KUKA KRL program: EPS_2_25716_MHCF01_A_20250828082512.src

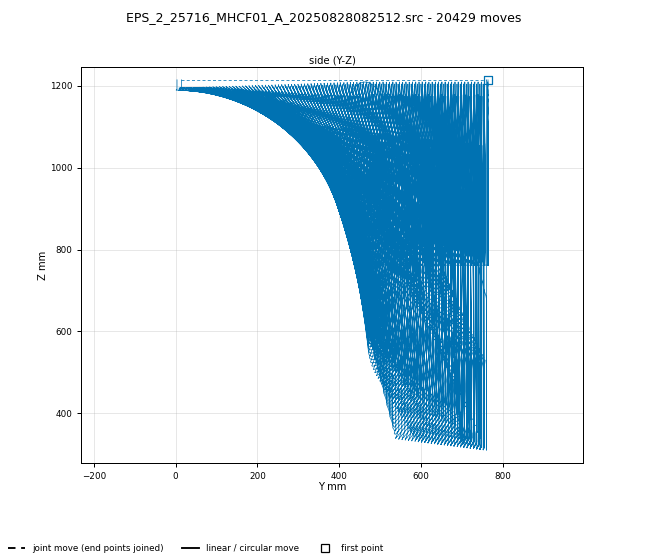
[picture p0: tool path of EPS_2_25716_MHCF01_A_20250828082512.src, 20429 of 20431 moves have a stored position in this frame; points joined in program order, loops and branches not executed]
&ACCESS RVP
&REL 4
&COMMENT QRS 19112012
&PARAM EDITMASK = *
DEF PART()
EXT BAS (BAS_COMMAND :IN,REAL :IN )
INT I
BAS (#INITMOV,0 )

;KUKA QRS Post kuka4.cps  Date:22-06-2017 !

File_ID=2800

QRS_PRE_INIT()

;Init var - Until changes are made in qrs_pre_init
Outlet_Square_prg=0
Inlet_1_Square_prg=0
Inlet_2_Square_prg=0
Inlet_3_Square_prg=0
Inlet_4_Square_prg=0
Inlet_5_Square_prg=0

Outlet_1={X 0.000, Y 457.000, Z 786.000, B 0.000, E1 0.000 }
Inlet_1={X 0.000, Y 688.000, Z 484.500, B 0.000, E1 109.000 }
Inlet_2={X 0.000, Y 457.000, Z 756.000, B 0.000, E1 180.000 }
Outlet_1_type=838
Inlet_1_type=201
Inlet_2_type=838
;QRS#1=Sidecore dimensions
;QRS#2=825-33" Concrete
;QRS#3=200-8" PVC SDR 35
;QRS#4=825-33" Concrete
;QRS#5=
;QRS#6=
;QRS#7=
;QRS#8=
;QRS#9=S306-46
;QRS#10=12-08 PSX
;QRS#11=S306-46
;QRS#12=
;QRS#13=
;QRS#14=
;QRS#15=
;QRS#16=1524x152x1676 5,5'
;QRS#17=EPS Height
;QRS#18=1205
;QRS#19=*
;QRS#20= UPDATED VERSION 22-06-2017
;QRS#21=*
Outlet_Square=0650
Inlet_1_Square=0100
Inlet_2_Square=0650
Inlet_3_Square=0
Inlet_4_Square=0
Inlet_5_Square=0
Mill_Square=1
Outlet_Square_Prg=267
Inlet_1_Square_prg=204
Inlet_2_Square_prg=267

QRS_INIT()

$ADVANCE=5

; T1
PTP {E1 176.359,E2 176.359}
PTP {X 0,Y 763.722,A -85,B 0,C 180,E1 176.359,E2 176.359,E3 0,E4 0,E5 0,E6 0}
QRS_SPEED_INIT()
LIN {X 0,Y 763.722,Z 1215,A -85,B 0,C 180,E1 176.359,E2 176.359,E3 0,E4 0,E5 0,E6 0} C_VEL
LIN {X 0,Y 763.722,Z 764.06,A -85,B 0,C 180,E1 176.359,E2 176.359} C_VEL
LIN {X 0,Y 763.74,Z 762.06,A -85,B 0,C 180,E1 176.509,E2 176.509} C_VEL
LIN {X 0,Y 763.887,Z 762.06,A -85,B 0,C 180,E1 177.187,E2 177.187} C_VEL
LIN {X 0,Y 763.859,Z 762.06,A -85,B 0,C 180,E1 184.692,E2 184.692} C_VEL
LIN {X 0,Y 763.829,Z 762.06,A -85,B 0,C 180,E1 192.28,E2 192.28} C_VEL
LIN {X 0,Y 763.844,Z 762.06,A -85,B 0,C 180,E1 200.095,E2 200.095} C_VEL
LIN {X 0,Y 763.817,Z 762.06,A -85,B 0,C 180,E1 208.325,E2 208.325} C_VEL
LIN {X 0,Y 762.405,Z 762.06,A -85,B 0,C 180,E1 210.54,E2 210.54} C_VEL
LIN {X 0,Y 762.716,Z 762.06,A -85,B 0,C 180,E1 214.993,E2 214.993} C_VEL
LIN {X 0,Y 763.716,Z 762.06,A -85,B 0,C 180,E1 216.696,E2 216.696} C_VEL
LIN {X 0,Y 763.502,Z 762.06,A -85,B 0,C 180,E1 224.735,E2 224.735} C_VEL
LIN {X 0,Y 763.769,Z 762.06,A -85,B 0,C 180,E1 225.284,E2 225.284} C_VEL
LIN {X 0,Y 763.693,Z 762.06,A -85,B 0,C 180,E1 233.306,E2 233.306} C_VEL
LIN {X 0,Y 763.603,Z 762.06,A -85,B 0,C 180,E1 233.585,E2 233.585} C_VEL
LIN {X 0,Y 763.11,Z 765.125,A -85,B 0,C 180,E1 233.691,E2 233.691} C_VEL
LIN {X 0,Y 763.161,Z 825.383,A -85,B 0,C 180,E1 234.39,E2 234.39} C_VEL
LIN {X 0,Y 763.585,Z 842.967,A -85,B 0,C 180,E1 234.683,E2 234.683} C_VEL
LIN {X 0,Y 763.687,Z 860.331,A -85,B 0,C 180,E1 235.017,E2 235.017} C_VEL
LIN {X 0,Y 763.614,Z 876.794,A -85,B 0,C 180,E1 235.382,E2 235.382} C_VEL
LIN {X 0,Y 763.265,Z 892.83,A -85,B 0,C 180,E1 235.785,E2 235.785} C_VEL
LIN {X 0,Y 763.632,Z 912.821,A -85,B 0,C 180,E1 236.407,E2 236.407} C_VEL
LIN {X 0,Y 763.653,Z 925.004,A -85,B 0,C 180,E1 236.825,E2 236.825} C_VEL
LIN {X 0,Y 763.67,Z 937.193,A -85,B 0,C 180,E1 237.266,E2 237.266} C_VEL
LIN {X 0,Y 763.647,Z 955.469,A -85,B 0,C 180,E1 238,E2 238} C_VEL
LIN {X 0,Y 763.481,Z 968.04,A -85,B 0,C 180,E1 238.551,E2 238.551} C_VEL
LIN {X 0,Y 763.562,Z 976.639,A -85,B 0,C 180,E1 238.958,E2 238.958} C_VEL
LIN {X 0,Y 763.516,Z 991.054,A -85,B 0,C 180,E1 239.67,E2 239.67} C_VEL
LIN {X 0,Y 763.481,Z 1008.327,A -85,B 0,C 180,E1 240.607,E2 240.607} C_VEL
LIN {X 0,Y 763.638,Z 1024.574,A -85,B 0,C 180,E1 241.577,E2 241.577} C_VEL
LIN {X 0,Y 763.597,Z 1040.363,A -85,B 0,C 180,E1 242.593,E2 242.593} C_VEL
LIN {X 0,Y 763.3,Z 1055.407,A -85,B 0,C 180,E1 243.633,E2 243.633} C_VEL
LIN {X 0,Y 763.19,Z 1070.044,A -85,B 0,C 180,E1 244.738,E2 244.738} C_VEL
LIN {X 0,Y 763.448,Z 1083.451,A -85,B 0,C 180,E1 245.843,E2 245.843} C_VEL
LIN {X 0,Y 763.685,Z 1096.507,A -85,B 0,C 180,E1 247.002,E2 247.002} C_VEL
LIN {X 0,Y 763.164,Z 1110.017,A -85,B 0,C 180,E1 248.281,E2 248.281} C_VEL
LIN {X 0,Y 762.922,Z 1121.794,A -85,B 0,C 180,E1 249.496,E2 249.496} C_VEL
LIN {X 0,Y 763.257,Z 1133.579,A -85,B 0,C 180,E1 250.838,E2 250.838} C_VEL
LIN {X 0,Y 763.827,Z 1143.997,A -85,B 0,C 180,E1 252.134,E2 252.134} C_VEL
LIN {X 0,Y 763.056,Z 1154.828,A -85,B 0,C 180,E1 253.589,E2 253.589} C_VEL
LIN {X 0,Y 762.742,Z 1164.591,A -85,B 0,C 180,E1 255.058,E2 255.058} C_VEL
LIN {X 0,Y 763.115,Z 1172.356,A -85,B 0,C 180,E1 256.36,E2 256.36} C_VEL
LIN {X 0,Y 763.85,Z 1179.543,A -85,B 0,C 180,E1 257.719,E2 257.719} C_VEL
LIN {X 0,Y 762.886,Z 1187.41,A -85,B 0,C 180,E1 259.379,E2 259.379} C_VEL
LIN {X 0,Y 762.625,Z 1192.228,A -85,B 0,C 180,E1 260.568,E2 260.568} C_VEL
LIN {X 0,Y 762.79,Z 1195.671,A -85,B 0,C 180,E1 261.52,E2 261.52} C_VEL
LIN {X 0,Y 763.28,Z 1198.709,A -85,B 0,C 180,E1 262.473,E2 262.473} C_VEL
LIN {X 0,Y 763.858,Z 1201.341,A -85,B 0,C 180,E1 263.423,E2 263.423} C_VEL
LIN {X 0,Y 763.267,Z 1203.655,A -85,B 0,C 180,E1 264.361,E2 264.361} C_VEL
LIN {X 0,Y 762.79,Z 1205.61,A -85,B 0,C 180,E1 265.3,E2 265.3} C_VEL
LIN {X 0,Y 762.61,Z 1207.2,A -85,B 0,C 180,E1 266.241,E2 266.241} C_VEL
LIN {X 0,Y 762.976,Z 1208.861,A -85,B 0,C 180,E1 267.626,E2 267.626} C_VEL
LIN {X 0,Y 763.872,Z 1209.666,A -85,B 0,C 180,E1 269.062,E2 269.062} C_VEL
LIN {X 0,Y 762.824,Z 1209.715,A -85,B 0,C 180,E1 270.938,E2 270.938} C_VEL
LIN {X 0,Y 762.626,Z 1209.464,A -85,B 0,C 180,E1 271.62,E2 271.62} C_VEL
LIN {X 0,Y 762.799,Z 1208.403,A -85,B 0,C 180,E1 272.816,E2 272.816} C_VEL
LIN {X 0,Y 763.271,Z 1207.186,A -85,B 0,C 180,E1 273.754,E2 273.754} C_VEL
LIN {X 0,Y 763.867,Z 1205.578,A -85,B 0,C 180,E1 274.691,E2 274.691} C_VEL
LIN {X 0,Y 763.013,Z 1202.59,A -85,B 0,C 180,E1 276.11,E2 276.11} C_VEL
LIN {X 0,Y 762.637,Z 1198.719,A -85,B 0,C 180,E1 277.532,E2 277.532} C_VEL
LIN {X 0,Y 762.799,Z 1195.679,A -85,B 0,C 180,E1 278.478,E2 278.478} C_VEL
LIN {X 0,Y 763.569,Z 1190.402,A -85,B 0,C 180,E1 279.894,E2 279.894} C_VEL
LIN {X 0,Y 763.864,Z 1188.414,A -85,B 0,C 180,E1 280.366,E2 280.366} C_VEL
LIN {X 0,Y 763.206,Z 1182.988,A -85,B 0,C 180,E1 281.57,E2 281.57} C_VEL
LIN {X 0,Y 762.859,Z 1179.555,A -85,B 0,C 180,E1 282.295,E2 282.295} C_VEL
LIN {X 0,Y 762.736,Z 1172.088,A -85,B 0,C 180,E1 283.694,E2 283.694} C_VEL
LIN {X 0,Y 763.29,Z 1163.914,A -85,B 0,C 180,E1 285.044,E2 285.044} C_VEL
LIN {X 0,Y 763.763,Z 1158.345,A -85,B 0,C 180,E1 285.87,E2 285.87} C_VEL
LIN {X 0,Y 763.637,Z 1154.843,A -85,B 0,C 180,E1 286.396,E2 286.396} C_VEL
LIN {X 0,Y 762.912,Z 1144.015,A -85,B 0,C 180,E1 287.885,E2 287.885} C_VEL
LIN {X 0,Y 762.868,Z 1131.999,A -85,B 0,C 180,E1 289.358,E2 289.358} C_VEL
LIN {X 0,Y 763.42,Z 1120.427,A -85,B 0,C 180,E1 290.638,E2 290.638} C_VEL
LIN {X 0,Y 763.768,Z 1112.188,A -85,B 0,C 180,E1 291.477,E2 291.477} C_VEL
LIN {X 0,Y 763.558,Z 1105.867,A -85,B 0,C 180,E1 292.112,E2 292.112} C_VEL
LIN {X 0,Y 763.217,Z 1095.124,A -85,B 0,C 180,E1 293.139,E2 293.139} C_VEL
LIN {X 0,Y 763.157,Z 1081.838,A -85,B 0,C 180,E1 294.303,E2 294.303} C_VEL
LIN {X 0,Y 763.464,Z 1068.233,A -85,B 0,C 180,E1 295.394,E2 295.394} C_VEL
LIN {X 0,Y 763.661,Z 1053.626,A -85,B 0,C 180,E1 296.482,E2 296.482} C_VEL
LIN {X 0,Y 763.464,Z 1037.389,A -85,B 0,C 180,E1 297.608,E2 297.608} C_VEL
LIN {X 0,Y 763.397,Z 1021.761,A -85,B 0,C 180,E1 298.604,E2 298.604} C_VEL
LIN {X 0,Y 763.561,Z 1005.354,A -85,B 0,C 180,E1 299.557,E2 299.557} C_VEL
LIN {X 0,Y 763.593,Z 989.474,A -85,B 0,C 180,E1 300.41,E2 300.41} C_VEL
LIN {X 0,Y 763.623,Z 970.492,A -85,B 0,C 180,E1 301.334,E2 301.334} C_VEL
LIN {X 0,Y 763.591,Z 951.717,A -85,B 0,C 180,E1 302.16,E2 302.16} C_VEL
LIN {X 0,Y 763.583,Z 933.277,A -85,B 0,C 180,E1 302.887,E2 302.887} C_VEL
LIN {X 0,Y 763.349,Z 920.518,A -85,B 0,C 180,E1 303.348,E2 303.348} C_VEL
LIN {X 0,Y 763.571,Z 911.94,A -85,B 0,C 180,E1 303.623,E2 303.623} C_VEL
LIN {X 0,Y 763.721,Z 893.155,A -85,B 0,C 180,E1 304.183,E2 304.183} C_VEL
LIN {X 0,Y 763.708,Z 877.523,A -85,B 0,C 180,E1 304.595,E2 304.595} C_VEL
LIN {X 0,Y 763.535,Z 860.886,A -85,B 0,C 180,E1 304.979,E2 304.979} C_VEL
LIN {X 0,Y 763.204,Z 848.058,A -85,B 0,C 180,E1 305.249,E2 305.249} C_VEL
LIN {X 0,Y 763.489,Z 831.034,A -85,B 0,C 180,E1 305.511,E2 305.511} C_VEL
LIN {X 0,Y 763.515,Z 819.053,A -85,B 0,C 180,E1 305.669,E2 305.669} C_VEL
LIN {X 0,Y 763.118,Z 762.451,A -85,B 0,C 180,E1 306.339,E2 306.339} C_VEL
LIN {X 0,Y 763.741,Z 762.06,A -85,B 0,C 180,E1 306.442,E2 306.442} C_VEL
LIN {X 0,Y 763.705,Z 762.06,A -85,B 0,C 180,E1 306.695,E2 306.695} C_VEL
LIN {X 0,Y 763.761,Z 762.06,A -85,B 0,C 180,E1 314.713,E2 314.713} C_VEL
LIN {X 0,Y 763.525,Z 762.06,A -85,B 0,C 180,E1 315.267,E2 315.267} C_VEL
LIN {X 0,Y 762.411,Z 762.06,A -85,B 0,C 180,E1 320.387,E2 320.387} C_VEL
LIN {X 0,Y 763.765,Z 762.06,A -85,B 0,C 180,E1 322.742,E2 322.742} C_VEL
LIN {X 0,Y 763.828,Z 762.06,A -85,B 0,C 180,E1 329.523,E2 329.523} C_VEL
LIN {X 0,Y 763.838,Z 762.06,A -85,B 0,C 180,E1 335.857,E2 335.857} C_VEL
LIN {X 0,Y 763.844,Z 762.06,A -85,B 0,C 180,E1 343.851,E2 343.851} C_VEL
LIN {X 0,Y 763.841,Z 762.06,A -85,B 0,C 180,E1 351.533,E2 351.533} C_VEL
LIN {X 0,Y 763.874,Z 762.06,A -85,B 0,C 180,E1 359.063,E2 359.063} C_VEL
LIN {X 0,Y 763.873,Z 762.06,A -85,B 0,C 180,E1 366.576,E2 366.576} C_VEL
LIN {X 0,Y 763.842,Z 762.06,A -85,B 0,C 180,E1 374.206,E2 374.206} C_VEL
LIN {X 0,Y 763.813,Z 762.06,A -85,B 0,C 180,E1 382.105,E2 382.105} C_VEL
LIN {X 0,Y 762.966,Z 762.06,A -85,B 0,C 180,E1 388.36,E2 388.36} C_VEL
LIN {X 0,Y 763.69,Z 762.06,A -85,B 0,C 180,E1 389.858,E2 389.858} C_VEL
LIN {X 0,Y 763.788,Z 762.06,A -85,B 0,C 180,E1 397.257,E2 397.257} C_VEL
LIN {X 0,Y 762.288,Z 762.06,A -85,B 0,C 180,E1 402.464,E2 402.464} C_VEL
LIN {X 0,Y 763.518,Z 762.06,A -85,B 0,C 180,E1 404.734,E2 404.734} C_VEL
LIN {X 0,Y 763.738,Z 762.06,A -85,B 0,C 180,E1 405.285,E2 405.285} C_VEL
LIN {X 0,Y 763.711,Z 762.06,A -85,B 0,C 180,E1 413.304,E2 413.304} C_VEL
LIN {X 0,Y 763.665,Z 762.06,A -85,B 0,C 180,E1 413.601,E2 413.601} C_VEL
LIN {X 0,Y 761.693,Z 762.06,A -85,B 0,C 180,E1 413.812,E2 413.812} C_VEL
LIN {X 0,Y 761.807,Z 763.834,A -85,B 0,C 180,E1 413.903,E2 413.903} C_VEL
LIN {X 0,Y 762.762,Z 766.677,A -85,B 0,C 180,E1 413.987,E2 413.987} C_VEL
LIN {X 0,Y 763.131,Z 768.605,A -85,B 0,C 180,E1 414.029,E2 414.029} C_VEL
LIN {X 0,Y 763.648,Z 798.138,A -85,B 0,C 180,E1 414.411,E2 414.411} C_VEL
LIN {X 0,Y 763.664,Z 815.21,A -85,B 0,C 180,E1 414.679,E2 414.679} C_VEL
LIN {X 0,Y 763.409,Z 832.281,A -85,B 0,C 180,E1 414.998,E2 414.998} C_VEL
LIN {X 0,Y 763.24,Z 839.694,A -85,B 0,C 180,E1 415.153,E2 415.153} C_VEL
LIN {X 0,Y 763.609,Z 855.772,A -85,B 0,C 180,E1 415.565,E2 415.565} C_VEL
LIN {X 0,Y 763.663,Z 868.895,A -85,B 0,C 180,E1 415.935,E2 415.935} C_VEL
LIN {X 0,Y 763.644,Z 887.88,A -85,B 0,C 180,E1 416.529,E2 416.529} C_VEL
LIN {X 0,Y 763.368,Z 905.889,A -85,B 0,C 180,E1 417.155,E2 417.155} C_VEL
LIN {X 0,Y 763.602,Z 925.254,A -85,B 0,C 180,E1 417.944,E2 417.944} C_VEL
LIN {X 0,Y 763.603,Z 943.443,A -85,B 0,C 180,E1 418.758,E2 418.758} C_VEL
LIN {X 0,Y 763.642,Z 961.593,A -85,B 0,C 180,E1 419.66,E2 419.66} C_VEL
LIN {X 0,Y 763.586,Z 977.603,A -85,B 0,C 180,E1 420.524,E2 420.524} C_VEL
LIN {X 0,Y 763.415,Z 994.185,A -85,B 0,C 180,E1 421.498,E2 421.498} C_VEL
LIN {X 0,Y 763.335,Z 1011.042,A -85,B 0,C 180,E1 422.585,E2 422.585} C_VEL
LIN {X 0,Y 763.547,Z 1026.034,A -85,B 0,C 180,E1 423.645,E2 423.645} C_VEL
LIN {X 0,Y 763.647,Z 1040.062,A -85,B 0,C 180,E1 424.711,E2 424.711} C_VEL
LIN {X 0,Y 763.256,Z 1053.988,A -85,B 0,C 180,E1 425.839,E2 425.839} C_VEL
LIN {X 0,Y 763.018,Z 1067.004,A -85,B 0,C 180,E1 426.983,E2 426.983} C_VEL
LIN {X 0,Y 763.297,Z 1080.095,A -85,B 0,C 180,E1 428.248,E2 428.248} C_VEL
LIN {X 0,Y 763.803,Z 1092.173,A -85,B 0,C 180,E1 429.518,E2 429.518} C_VEL
LIN {X 0,Y 763.199,Z 1103.736,A -85,B 0,C 180,E1 430.811,E2 430.811} C_VEL
LIN {X 0,Y 762.791,Z 1114.347,A -85,B 0,C 180,E1 432.112,E2 432.112} C_VEL
LIN {X 0,Y 763.102,Z 1125.142,A -85,B 0,C 180,E1 433.592,E2 433.592} C_VEL
LIN {X 0,Y 763.761,Z 1133.68,A -85,B 0,C 180,E1 434.882,E2 434.882} C_VEL
LIN {X 0,Y 763.673,Z 1136.311,A -85,B 0,C 180,E1 435.318,E2 435.318} C_VEL
LIN {X 0,Y 762.988,Z 1143.295,A -85,B 0,C 180,E1 436.488,E2 436.488} C_VEL
LIN {X 0,Y 762.6,Z 1150.963,A -85,B 0,C 180,E1 437.941,E2 437.941} C_VEL
LIN {X 0,Y 763.021,Z 1157.607,A -85,B 0,C 180,E1 439.383,E2 439.383} C_VEL
LIN {X 0,Y 763.734,Z 1162.407,A -85,B 0,C 180,E1 440.584,E2 440.584} C_VEL
LIN {X 0,Y 763.71,Z 1164.155,A -85,B 0,C 180,E1 441.058,E2 441.058} C_VEL
LIN {X 0,Y 763.145,Z 1167.372,A -85,B 0,C 180,E1 442,E2 442} C_VEL
LIN {X 0,Y 762.743,Z 1170.222,A -85,B 0,C 180,E1 442.943,E2 442.943} C_VEL
LIN {X 0,Y 762.645,Z 1172.699,A -85,B 0,C 180,E1 443.887,E2 443.887} C_VEL
LIN {X 0,Y 763.158,Z 1175.695,A -85,B 0,C 180,E1 445.305,E2 445.305} C_VEL
LIN {X 0,Y 763.838,Z 1177.41,A -85,B 0,C 180,E1 446.389,E2 446.389} C_VEL
LIN {X 0,Y 763.399,Z 1178.43,A -85,B 0,C 180,E1 447.186,E2 447.186} C_VEL
LIN {X 0,Y 762.558,Z 1179.735,A -85,B 0,C 180,E1 449.062,E2 449.062} C_VEL
LIN {X 0,Y 762.983,Z 1179.696,A -85,B 0,C 180,E1 450.94,E2 450.94} C_VEL
LIN {X 0,Y 763.578,Z 1178.326,A -85,B 0,C 180,E1 452.815,E2 452.815} C_VEL
LIN {X 0,Y 763.007,Z 1177.129,A -85,B 0,C 180,E1 453.757,E2 453.757} C_VEL
LIN {X 0,Y 762.687,Z 1175.523,A -85,B 0,C 180,E1 454.7,E2 454.7} C_VEL
LIN {X 0,Y 762.806,Z 1172.471,A -85,B 0,C 180,E1 456.114,E2 456.114} C_VEL
LIN {X 0,Y 763.563,Z 1168.572,A -85,B 0,C 180,E1 457.525,E2 457.525} C_VEL
LIN {X 0,Y 763.871,Z 1167.062,A -85,B 0,C 180,E1 457.994,E2 457.994} C_VEL
LIN {X 0,Y 763.298,Z 1163.834,A -85,B 0,C 180,E1 458.949,E2 458.949} C_VEL
LIN {X 0,Y 762.809,Z 1160.211,A -85,B 0,C 180,E1 459.906,E2 459.906} C_VEL
LIN {X 0,Y 762.632,Z 1156.118,A -85,B 0,C 180,E1 460.863,E2 460.863} C_VEL
LIN {X 0,Y 763.012,Z 1149.302,A -85,B 0,C 180,E1 462.295,E2 462.295} C_VEL
LIN {X 0,Y 763.742,Z 1142.426,A -85,B 0,C 180,E1 463.571,E2 463.571} C_VEL
LIN {X 0,Y 763.77,Z 1140.524,A -85,B 0,C 180,E1 463.889,E2 463.889} C_VEL
LIN {X 0,Y 763.149,Z 1133.842,A -85,B 0,C 180,E1 465.014,E2 465.014} C_VEL
LIN {X 0,Y 762.72,Z 1124.527,A -85,B 0,C 180,E1 466.419,E2 466.419} C_VEL
LIN {X 0,Y 763.111,Z 1112.649,A -85,B 0,C 180,E1 468.006,E2 468.006} C_VEL
LIN {X 0,Y 763.786,Z 1101.998,A -85,B 0,C 180,E1 469.289,E2 469.289} C_VEL
LIN {X 0,Y 763.295,Z 1090.039,A -85,B 0,C 180,E1 470.636,E2 470.636} C_VEL
LIN {X 0,Y 762.981,Z 1078.156,A -85,B 0,C 180,E1 471.867,E2 471.867} C_VEL
LIN {X 0,Y 763.239,Z 1064.584,A -85,B 0,C 180,E1 473.14,E2 473.14} C_VEL
LIN {X 0,Y 763.68,Z 1051.16,A -85,B 0,C 180,E1 474.295,E2 474.295} C_VEL
LIN {X 0,Y 763.565,Z 1039.109,A -85,B 0,C 180,E1 475.278,E2 475.278} C_VEL
LIN {X 0,Y 763.278,Z 1022.943,A -85,B 0,C 180,E1 476.498,E2 476.498} C_VEL
LIN {X 0,Y 763.364,Z 1007.682,A -85,B 0,C 180,E1 477.548,E2 477.548} C_VEL
LIN {X 0,Y 763.578,Z 991.976,A -85,B 0,C 180,E1 478.539,E2 478.539} C_VEL
LIN {X 0,Y 763.634,Z 974.917,A -85,B 0,C 180,E1 479.532,E2 479.532} C_VEL
LIN {X 0,Y 763.542,Z 958.559,A -85,B 0,C 180,E1 480.413,E2 480.413} C_VEL
LIN {X 0,Y 763.571,Z 940.113,A -85,B 0,C 180,E1 481.309,E2 481.309} C_VEL
LIN {X 0,Y 763.536,Z 921.233,A -85,B 0,C 180,E1 482.137,E2 482.137} C_VEL
LIN {X 0,Y 763.431,Z 914.252,A -85,B 0,C 180,E1 482.419,E2 482.419} C_VEL
LIN {X 0,Y 763.666,Z 902.086,A -85,B 0,C 180,E1 482.879,E2 482.879} C_VEL
LIN {X 0,Y 763.698,Z 884.096,A -85,B 0,C 180,E1 483.505,E2 483.505} C_VEL
LIN {X 0,Y 763.64,Z 863.566,A -85,B 0,C 180,E1 484.131,E2 484.131} C_VEL
LIN {X 0,Y 763.324,Z 846.79,A -85,B 0,C 180,E1 484.588,E2 484.588} C_VEL
LIN {X 0,Y 763.327,Z 841.786,A -85,B 0,C 180,E1 484.704,E2 484.704} C_VEL
LIN {X 0,Y 763.694,Z 825.562,A -85,B 0,C 180,E1 485.036,E2 485.036} C_VEL
LIN {X 0,Y 763.758,Z 807.93,A -85,B 0,C 180,E1 485.347,E2 485.347} C_VEL
LIN {X 0,Y 763.695,Z 792.713,A -85,B 0,C 180,E1 485.569,E2 485.569} C_VEL
LIN {X 0,Y 763.223,Z 767.95,A -85,B 0,C 180,E1 485.883,E2 485.883} C_VEL
LIN {X 0,Y 763.265,Z 762.06,A -85,B 0,C 180,E1 485.98,E2 485.98} C_VEL
LIN {X 0,Y 763.595,Z 762.06,A -85,B 0,C 180,E1 486.6,E2 486.6} C_VEL
LIN {X 0,Y 763.808,Z 762.06,A -85,B 0,C 180,E1 492.131,E2 492.131} C_VEL
LIN {X 0,Y 763.614,Z 762.06,A -85,B 0,C 180,E1 492.57,E2 492.57} C_VEL
LIN {X 0,Y 763.875,Z 762.06,A -85,B 0,C 180,E1 500.258,E2 500.258} C_VEL
LIN {X 0,Y 763.733,Z 762.06,A -85,B 0,C 180,E1 506.566,E2 506.566} C_VEL
LIN {X 0,Y 763.499,Z 762.06,A -85,B 0,C 180,E1 507.306,E2 507.306} C_VEL
LIN {X 0,Y 763.209,Z 762.122,A -85,B 0,C 180,E1 507.486,E2 507.486} C_VEL
LIN {X 0,Y 763.638,Z 763.12,A -85,B 0,C 180,E1 507.53,E2 507.53} C_VEL
LIN {X 0,Y 763.79,Z 765.738,A -85,B 0,C 180,E1 507.626,E2 507.626} C_VEL
LIN {X 0,Y 763.797,Z 831.68,A -85,B 0,C 180,E1 509.978,E2 509.978} C_VEL
LIN {X 0,Y 763.29,Z 835.99,A -85,B 0,C 180,E1 510.124,E2 510.124} C_VEL
LIN {X 0,Y 763.012,Z 837.649,A -85,B 0,C 180,E1 510.172,E2 510.172} C_VEL
LIN {X 0,Y 763.701,Z 916.034,A -85,B 0,C 180,E1 510.916,E2 510.916} C_VEL
LIN {X 0,Y 763.838,Z 948.168,A -85,B 0,C 180,E1 511.225,E2 511.225} C_VEL
LIN {X 0,Y 763.826,Z 957.76,A -85,B 0,C 180,E1 511.354,E2 511.354} C_VEL
LIN {X 0,Y 763.852,Z 968.842,A -85,B 0,C 180,E1 511.58,E2 511.58} C_VEL
LIN {X 0,Y 763.85,Z 979.495,A -85,B 0,C 180,E1 511.875,E2 511.875} C_VEL
LIN {X 0,Y 763.751,Z 990.547,A -85,B 0,C 180,E1 512.269,E2 512.269} C_VEL
LIN {X 0,Y 763.666,Z 1000.84,A -85,B 0,C 180,E1 512.728,E2 512.728} C_VEL
LIN {X 0,Y 763.853,Z 1010.575,A -85,B 0,C 180,E1 513.262,E2 513.262} C_VEL
LIN {X 0,Y 763.738,Z 1018.552,A -85,B 0,C 180,E1 513.781,E2 513.781} C_VEL
LIN {X 0,Y 763.337,Z 1026.8,A -85,B 0,C 180,E1 514.414,E2 514.414} C_VEL
LIN {X 0,Y 763.391,Z 1034.378,A -85,B 0,C 180,E1 515.117,E2 515.117} C_VEL
LIN {X 0,Y 763.816,Z 1040.943,A -85,B 0,C 180,E1 515.856,E2 515.856} C_VEL
LIN {X 0,Y 763.73,Z 1044.687,A -85,B 0,C 180,E1 516.366,E2 516.366} C_VEL
LIN {X 0,Y 763.556,Z 1046.498,A -85,B 0,C 180,E1 516.616,E2 516.616} C_VEL
LIN {X 0,Y 763.126,Z 1051.588,A -85,B 0,C 180,E1 517.493,E2 517.493} C_VEL
LIN {X 0,Y 763.403,Z 1055.387,A -85,B 0,C 180,E1 518.38,E2 518.38} C_VEL
LIN {X 0,Y 763.87,Z 1057.915,A -85,B 0,C 180,E1 519.233,E2 519.233} C_VEL
LIN {X 0,Y 763.413,Z 1059.478,A -85,B 0,C 180,E1 520.109,E2 520.109} C_VEL
LIN {X 0,Y 763.251,Z 1059.957,A -85,B 0,C 180,E1 521.032,E2 521.032} C_VEL
LIN {X 0,Y 763.655,Z 1059.354,A -85,B 0,C 180,E1 521.885,E2 521.885} C_VEL
LIN {X 0,Y 763.862,Z 1058.461,A -85,B 0,C 180,E1 522.382,E2 522.382} C_VEL
LIN {X 0,Y 763.738,Z 1058.034,A -85,B 0,C 180,E1 522.625,E2 522.625} C_VEL
LIN {X 0,Y 763.24,Z 1055.162,A -85,B 0,C 180,E1 523.594,E2 523.594} C_VEL
LIN {X 0,Y 763.303,Z 1051.925,A -85,B 0,C 180,E1 524.344,E2 524.344} C_VEL
LIN {X 0,Y 763.727,Z 1047.737,A -85,B 0,C 180,E1 525.09,E2 525.09} C_VEL
LIN {X 0,Y 763.841,Z 1046.258,A -85,B 0,C 180,E1 525.326,E2 525.326} C_VEL
LIN {X 0,Y 763.734,Z 1040.569,A -85,B 0,C 180,E1 526.099,E2 526.099} C_VEL
LIN {X 0,Y 763.771,Z 1035.105,A -85,B 0,C 180,E1 526.714,E2 526.714} C_VEL
LIN {X 0,Y 763.809,Z 1027.112,A -85,B 0,C 180,E1 527.466,E2 527.466} C_VEL
LIN {X 0,Y 763.493,Z 1019.373,A -85,B 0,C 180,E1 528.074,E2 528.074} C_VEL
LIN {X 0,Y 763.527,Z 1010.215,A -85,B 0,C 180,E1 528.673,E2 528.673} C_VEL
LIN {X 0,Y 763.845,Z 1000.103,A -85,B 0,C 180,E1 529.215,E2 529.215} C_VEL
LIN {X 0,Y 763.796,Z 989.571,A -85,B 0,C 180,E1 529.678,E2 529.678} C_VEL
LIN {X 0,Y 763.682,Z 979.025,A -85,B 0,C 180,E1 530.051,E2 530.051} C_VEL
LIN {X 0,Y 763.841,Z 967.337,A -85,B 0,C 180,E1 530.364,E2 530.364} C_VEL
LIN {X 0,Y 763.864,Z 955.826,A -85,B 0,C 180,E1 530.586,E2 530.586} C_VEL
LIN {X 0,Y 763.864,Z 944.689,A -85,B 0,C 180,E1 530.724,E2 530.724} C_VEL
LIN {X 0,Y 763.795,Z 840.857,A -85,B 0,C 180,E1 531.697,E2 531.697} C_VEL
LIN {X 0,Y 763.395,Z 837.234,A -85,B 0,C 180,E1 531.74,E2 531.74} C_VEL
LIN {X 0,Y 763.377,Z 762.06,A -85,B 0,C 180,E1 534.427,E2 534.427} C_VEL
LIN {X 0,Y 763.879,Z 762.06,A -85,B 0,C 180,E1 534.598,E2 534.598} C_VEL
LIN {X 0,Y 763.74,Z 762.06,A -85,B 0,C 180,E1 536.509,E2 536.509} C_VEL
LIN {X 0,Y 754.649,Z 762.06,A -85,B 0,C 180,E1 539.103,E2 539.103} C_VEL
LIN {X 0,Y 754.714,Z 762.06,A -85,B 0,C 180,E1 546.382,E2 546.382} C_VEL
LIN {X 0,Y 754.951,Z 762.06,A -85,B 0,C 180,E1 553.398,E2 553.398} C_VEL
LIN {X 0,Y 755.106,Z 762.06,A -85,B 0,C 180,E1 560.956,E2 560.956} C_VEL
LIN {X 0,Y 754.907,Z 762.06,A -85,B 0,C 180,E1 569.538,E2 569.538} C_VEL
LIN {X 0,Y 754.747,Z 762.06,A -85,B 0,C 180,E1 577.859,E2 577.859} C_VEL
LIN {X 0,Y 755.038,Z 762.06,A -85,B 0,C 180,E1 586.149,E2 586.149} C_VEL
LIN {X 0,Y 755.772,Z 763.476,A -85,B 0,C 180,E1 593.262,E2 593.262} C_VEL
LIN {X 0,Y 757.071,Z 866.865,A -85,B 0,C 180,E1 594.806,E2 594.806} C_VEL
LIN {X 0,Y 756.764,Z 937.982,A -85,B 0,C 180,E1 596.961,E2 596.961} C_VEL
LIN {X 0,Y 756.208,Z 1009.087,A -85,B 0,C 180,E1 600.342,E2 600.342} C_VEL
LIN {X 0,Y 755.591,Z 1073.769,A -85,B 0,C 180,E1 604.774,E2 604.774} C_VEL
LIN {X 0,Y 755.159,Z 1125.985,A -85,B 0,C 180,E1 609.753,E2 609.753} C_VEL
LIN {X 0,Y 754.885,Z 1162.64,A -85,B 0,C 180,E1 614.586,E2 614.586} C_VEL
LIN {X 0,Y 754.929,Z 1187.619,A -85,B 0,C 180,E1 619.317,E2 619.317} C_VEL
LIN {X 0,Y 755.011,Z 1204.817,A -85,B 0,C 180,E1 624.842,E2 624.842} C_VEL
LIN {X 0,Y 755.6,Z 1209.848,A -85,B 0,C 180,E1 629.455,E2 629.455} C_VEL
LIN {X 0,Y 755.213,Z 1203.673,A -85,B 0,C 180,E1 635.696,E2 635.696} C_VEL
LIN {X 0,Y 755.209,Z 1183.325,A -85,B 0,C 180,E1 641.622,E2 641.622} C_VEL
LIN {X 0,Y 755.279,Z 1149.721,A -85,B 0,C 180,E1 647.293,E2 647.293} C_VEL
LIN {X 0,Y 755.616,Z 1101.536,A -85,B 0,C 180,E1 652.773,E2 652.773} C_VEL
LIN {X 0,Y 756.053,Z 1041.761,A -85,B 0,C 180,E1 657.605,E2 657.605} C_VEL
LIN {X 0,Y 756.539,Z 972.654,A -85,B 0,C 180,E1 661.561,E2 661.561} C_VEL
LIN {X 0,Y 756.981,Z 899.217,A -85,B 0,C 180,E1 664.352,E2 664.352} C_VEL
LIN {X 0,Y 757.033,Z 825.171,A -85,B 0,C 180,E1 665.945,E2 665.945} C_VEL
LIN {X 0,Y 755.604,Z 762.06,A -85,B 0,C 180,E1 666.801,E2 666.801} C_VEL
LIN {X 0,Y 754.964,Z 762.06,A -85,B 0,C 180,E1 676.058,E2 676.058} C_VEL
LIN {X 0,Y 755.187,Z 762.06,A -85,B 0,C 180,E1 683.61,E2 683.61} C_VEL
LIN {X 0,Y 754.991,Z 762.06,A -85,B 0,C 180,E1 691.018,E2 691.018} C_VEL
LIN {X 0,Y 754.99,Z 762.06,A -85,B 0,C 180,E1 696.892,E2 696.892} C_VEL
LIN {X 0,Y 755.509,Z 762.06,A -85,B 0,C 180,E1 704.234,E2 704.234} C_VEL
LIN {X 0,Y 755.149,Z 762.06,A -85,B 0,C 180,E1 712.462,E2 712.462} C_VEL
LIN {X 0,Y 754.843,Z 762.06,A -85,B 0,C 180,E1 720.542,E2 720.542} C_VEL
LIN {X 0,Y 755.16,Z 762.06,A -85,B 0,C 180,E1 727.47,E2 727.47} C_VEL
LIN {X 0,Y 754.722,Z 762.06,A -85,B 0,C 180,E1 735.712,E2 735.712} C_VEL
LIN {X 0,Y 755.109,Z 762.06,A -85,B 0,C 180,E1 743.031,E2 743.031} C_VEL
LIN {X 0,Y 754.738,Z 762.06,A -85,B 0,C 180,E1 751.245,E2 751.245} C_VEL
LIN {X 0,Y 755.372,Z 762.06,A -85,B 0,C 180,E1 757.737,E2 757.737} C_VEL
LIN {X 0,Y 755.086,Z 762.06,A -85,B 0,C 180,E1 766.068,E2 766.068} C_VEL
LIN {X 0,Y 754.847,Z 762.617,A -85,B 0,C 180,E1 773.503,E2 773.503} C_VEL
LIN {X 0,Y 756.838,Z 851.222,A -85,B 0,C 180,E1 775.096,E2 775.096} C_VEL
LIN {X 0,Y 756.572,Z 927.019,A -85,B 0,C 180,E1 777.689,E2 777.689} C_VEL
LIN {X 0,Y 756.03,Z 997.6,A -85,B 0,C 180,E1 781.416,E2 781.416} C_VEL
LIN {X 0,Y 755.498,Z 1059.465,A -85,B 0,C 180,E1 786.063,E2 786.063} C_VEL
LIN {X 0,Y 755.207,Z 1107.459,A -85,B 0,C 180,E1 791.064,E2 791.064} C_VEL
LIN {X 0,Y 755.121,Z 1143.123,A -85,B 0,C 180,E1 796.312,E2 796.312} C_VEL
LIN {X 0,Y 755.209,Z 1167.271,A -85,B 0,C 180,E1 801.884,E2 801.884} C_VEL
LIN {X 0,Y 755.441,Z 1178.391,A -85,B 0,C 180,E1 807.091,E2 807.091} C_VEL
LIN {X 0,Y 755.577,Z 1178.361,A -85,B 0,C 180,E1 812.847,E2 812.847} C_VEL
LIN {X 0,Y 755.337,Z 1164.251,A -85,B 0,C 180,E1 818.926,E2 818.926} C_VEL
LIN {X 0,Y 755.313,Z 1136.006,A -85,B 0,C 180,E1 824.809,E2 824.809} C_VEL
LIN {X 0,Y 755.571,Z 1094.24,A -85,B 0,C 180,E1 830.389,E2 830.389} C_VEL
LIN {X 0,Y 755.949,Z 1039.354,A -85,B 0,C 180,E1 835.532,E2 835.532} C_VEL
LIN {X 0,Y 756.379,Z 973.926,A -85,B 0,C 180,E1 839.899,E2 839.899} C_VEL
LIN {X 0,Y 756.794,Z 902.312,A -85,B 0,C 180,E1 843.209,E2 843.209} C_VEL
LIN {X 0,Y 757.059,Z 828.537,A -85,B 0,C 180,E1 845.328,E2 845.328} C_VEL
LIN {X 0,Y 755.501,Z 762.06,A -85,B 0,C 180,E1 846.417,E2 846.417} C_VEL
LIN {X 0,Y 754.691,Z 762.06,A -85,B 0,C 180,E1 853.876,E2 853.876} C_VEL
LIN {X 0,Y 755.508,Z 762.06,A -85,B 0,C 180,E1 860.801,E2 860.801} C_VEL
LIN {X 0,Y 755.399,Z 762.845,A -85,B 0,C 180,E1 867.37,E2 867.37} C_VEL
LIN {X 0,Y 755.203,Z 841.66,A -85,B 0,C 180,E1 870.097,E2 870.097} C_VEL
LIN {X 0,Y 755.975,Z 969.088,A -85,B 0,C 180,E1 871.489,E2 871.489} C_VEL
LIN {X 0,Y 755.852,Z 1007.886,A -85,B 0,C 180,E1 873.027,E2 873.027} C_VEL
LIN {X 0,Y 755.636,Z 1038.476,A -85,B 0,C 180,E1 875.515,E2 875.515} C_VEL
LIN {X 0,Y 755.532,Z 1056.178,A -85,B 0,C 180,E1 878.603,E2 878.603} C_VEL
LIN {X 0,Y 755.659,Z 1059.384,A -85,B 0,C 180,E1 881.903,E2 881.903} C_VEL
LIN {X 0,Y 755.786,Z 1047.355,A -85,B 0,C 180,E1 885.205,E2 885.205} C_VEL
LIN {X 0,Y 755.593,Z 1021.178,A -85,B 0,C 180,E1 888.01,E2 888.01} C_VEL
LIN {X 0,Y 755.835,Z 985.532,A -85,B 0,C 180,E1 889.918,E2 889.918} C_VEL
LIN {X 0,Y 755.981,Z 944.278,A -85,B 0,C 180,E1 890.831,E2 890.831} C_VEL
LIN {X 0,Y 755.464,Z 831.48,A -85,B 0,C 180,E1 892.061,E2 892.061} C_VEL
LIN {X 0,Y 755.867,Z 762.06,A -85,B 0,C 180,E1 894.707,E2 894.707} C_VEL
LIN {X 0,Y 754.649,Z 762.06,A -85,B 0,C 180,E1 899.103,E2 899.103} C_VEL
LIN {X 0,Y 746.34,Z 762.06,A -85,B 0,C 180,E1 901.736,E2 901.736} C_VEL
LIN {X 0,Y 746.674,Z 762.06,A -85,B 0,C 180,E1 906.451,E2 906.451} C_VEL
LIN {X 0,Y 746.854,Z 762.06,A -85,B 0,C 180,E1 913.546,E2 913.546} C_VEL
LIN {X 0,Y 747.186,Z 762.06,A -85,B 0,C 180,E1 920.852,E2 920.852} C_VEL
LIN {X 0,Y 747.493,Z 762.06,A -85,B 0,C 180,E1 928.528,E2 928.528} C_VEL
LIN {X 0,Y 747.254,Z 762.06,A -85,B 0,C 180,E1 936.839,E2 936.839} C_VEL
LIN {X 0,Y 746.997,Z 762.06,A -85,B 0,C 180,E1 946.191,E2 946.191} C_VEL
LIN {X 0,Y 747.444,Z 763.808,A -85,B 0,C 180,E1 952.788,E2 952.788} C_VEL
LIN {X 0,Y 750.231,Z 776.864,A -85,B 0,C 180,E1 953.103,E2 953.103} C_VEL
LIN {X 0,Y 750.506,Z 865.678,A -85,B 0,C 180,E1 954.425,E2 954.425} C_VEL
LIN {X 0,Y 749.923,Z 935.971,A -85,B 0,C 180,E1 956.538,E2 956.538} C_VEL
LIN {X 0,Y 748.996,Z 1006.584,A -85,B 0,C 180,E1 959.878,E2 959.878} C_VEL
LIN {X 0,Y 748.022,Z 1071.537,A -85,B 0,C 180,E1 964.313,E2 964.313} C_VEL
LIN {X 0,Y 747.303,Z 1123.291,A -85,B 0,C 180,E1 969.22,E2 969.22} C_VEL
LIN {X 0,Y 747.011,Z 1160.66,A -85,B 0,C 180,E1 974.117,E2 974.117} C_VEL
LIN {X 0,Y 746.988,Z 1187.62,A -85,B 0,C 180,E1 979.202,E2 979.202} C_VEL
LIN {X 0,Y 747.047,Z 1204.817,A -85,B 0,C 180,E1 984.787,E2 984.787} C_VEL
LIN {X 0,Y 747.593,Z 1209.85,A -85,B 0,C 180,E1 989.449,E2 989.449} C_VEL
LIN {X 0,Y 747.473,Z 1204.698,A -85,B 0,C 180,E1 995.272,E2 995.272} C_VEL
LIN {X 0,Y 747.343,Z 1184.684,A -85,B 0,C 180,E1 1001.449,E2 1001.449} C_VEL
LIN {X 0,Y 747.377,Z 1150.917,A -85,B 0,C 180,E1 1007.317,E2 1007.317} C_VEL
LIN {X 0,Y 747.89,Z 1102.898,A -85,B 0,C 180,E1 1012.889,E2 1012.889} C_VEL
LIN {X 0,Y 748.614,Z 1043.481,A -85,B 0,C 180,E1 1017.781,E2 1017.781} C_VEL
LIN {X 0,Y 749.445,Z 974.583,A -85,B 0,C 180,E1 1021.798,E2 1021.798} C_VEL
LIN {X 0,Y 750.189,Z 902.678,A -85,B 0,C 180,E1 1024.598,E2 1024.598} C_VEL
LIN {X 0,Y 750.501,Z 828.692,A -85,B 0,C 180,E1 1026.256,E2 1026.256} C_VEL
LIN {X 0,Y 748.648,Z 766.444,A -85,B 0,C 180,E1 1027.111,E2 1027.111} C_VEL
LIN {X 0,Y 747.086,Z 762.06,A -85,B 0,C 180,E1 1027.435,E2 1027.435} C_VEL
LIN {X 0,Y 746.891,Z 762.06,A -85,B 0,C 180,E1 1036.198,E2 1036.198} C_VEL
LIN {X 0,Y 746.758,Z 762.06,A -85,B 0,C 180,E1 1044.574,E2 1044.574} C_VEL
LIN {X 0,Y 746.854,Z 762.06,A -85,B 0,C 180,E1 1051.445,E2 1051.445} C_VEL
LIN {X 0,Y 746.526,Z 762.06,A -85,B 0,C 180,E1 1057.72,E2 1057.72} C_VEL
LIN {X 0,Y 746.822,Z 762.06,A -85,B 0,C 180,E1 1065.253,E2 1065.253} C_VEL
LIN {X 0,Y 747.172,Z 762.06,A -85,B 0,C 180,E1 1072.381,E2 1072.381} C_VEL
LIN {X 0,Y 746.857,Z 762.06,A -85,B 0,C 180,E1 1080.548,E2 1080.548} C_VEL
LIN {X 0,Y 747.097,Z 762.06,A -85,B 0,C 180,E1 1087.551,E2 1087.551} C_VEL
LIN {X 0,Y 747.089,Z 762.06,A -85,B 0,C 180,E1 1095.146,E2 1095.146} C_VEL
LIN {X 0,Y 746.946,Z 762.06,A -85,B 0,C 180,E1 1103.297,E2 1103.297} C_VEL
LIN {X 0,Y 746.794,Z 762.06,A -85,B 0,C 180,E1 1111.164,E2 1111.164} C_VEL
LIN {X 0,Y 746.849,Z 762.06,A -85,B 0,C 180,E1 1118.489,E2 1118.489} C_VEL
LIN {X 0,Y 747.06,Z 762.06,A -85,B 0,C 180,E1 1126.087,E2 1126.087} C_VEL
LIN {X 0,Y 747.766,Z 763.987,A -85,B 0,C 180,E1 1133.117,E2 1133.117} C_VEL
LIN {X 0,Y 750.587,Z 792.853,A -85,B 0,C 180,E1 1133.623,E2 1133.623} C_VEL
LIN {X 0,Y 750.25,Z 865.72,A -85,B 0,C 180,E1 1135.143,E2 1135.143} C_VEL
LIN {X 0,Y 749.515,Z 936.849,A -85,B 0,C 180,E1 1137.796,E2 1137.796} C_VEL
LIN {X 0,Y 748.585,Z 1005.86,A -85,B 0,C 180,E1 1141.649,E2 1141.649} C_VEL
LIN {X 0,Y 747.69,Z 1066.56,A -85,B 0,C 180,E1 1146.441,E2 1146.441} C_VEL
LIN {X 0,Y 747.167,Z 1112.549,A -85,B 0,C 180,E1 1151.492,E2 1151.492} C_VEL
LIN {X 0,Y 747.055,Z 1144.678,A -85,B 0,C 180,E1 1156.461,E2 1156.461} C_VEL
LIN {X 0,Y 747.273,Z 1167.268,A -85,B 0,C 180,E1 1161.797,E2 1161.797} C_VEL
LIN {X 0,Y 747.441,Z 1178.391,A -85,B 0,C 180,E1 1167.06,E2 1167.06} C_VEL
LIN {X 0,Y 747.546,Z 1178.362,A -85,B 0,C 180,E1 1172.878,E2 1172.878} C_VEL
LIN {X 0,Y 747.284,Z 1164.254,A -85,B 0,C 180,E1 1179.022,E2 1179.022} C_VEL
LIN {X 0,Y 747.355,Z 1136.677,A -85,B 0,C 180,E1 1184.857,E2 1184.857} C_VEL
LIN {X 0,Y 747.764,Z 1095.593,A -85,B 0,C 180,E1 1190.456,E2 1190.456} C_VEL
LIN {X 0,Y 748.338,Z 1040.471,A -85,B 0,C 180,E1 1195.72,E2 1195.72} C_VEL
LIN {X 0,Y 749.131,Z 975.529,A -85,B 0,C 180,E1 1200.13,E2 1200.13} C_VEL
LIN {X 0,Y 749.918,Z 903.828,A -85,B 0,C 180,E1 1203.498,E2 1203.498} C_VEL
LIN {X 0,Y 750.478,Z 829.13,A -85,B 0,C 180,E1 1205.673,E2 1205.673} C_VEL
LIN {X 0,Y 748.696,Z 766.238,A -85,B 0,C 180,E1 1206.713,E2 1206.713} C_VEL
LIN {X 0,Y 747.354,Z 762.06,A -85,B 0,C 180,E1 1207.061,E2 1207.061} C_VEL
LIN {X 0,Y 746.682,Z 762.06,A -85,B 0,C 180,E1 1213.883,E2 1213.883} C_VEL
LIN {X 0,Y 747,Z 762.06,A -85,B 0,C 180,E1 1221.764,E2 1221.764} C_VEL
LIN {X 0,Y 747.616,Z 763.311,A -85,B 0,C 180,E1 1227.243,E2 1227.243} C_VEL
LIN {X 0,Y 747.365,Z 841.333,A -85,B 0,C 180,E1 1229.978,E2 1229.978} C_VEL
LIN {X 0,Y 748.082,Z 969.974,A -85,B 0,C 180,E1 1231.411,E2 1231.411} C_VEL
LIN {X 0,Y 747.902,Z 1008.335,A -85,B 0,C 180,E1 1232.966,E2 1232.966} C_VEL
LIN {X 0,Y 747.618,Z 1038.455,A -85,B 0,C 180,E1 1235.453,E2 1235.453} C_VEL
LIN {X 0,Y 747.427,Z 1055.433,A -85,B 0,C 180,E1 1238.332,E2 1238.332} C_VEL
LIN {X 0,Y 747.573,Z 1059.601,A -85,B 0,C 180,E1 1241.7,E2 1241.7} C_VEL
LIN {X 0,Y 747.64,Z 1049.145,A -85,B 0,C 180,E1 1244.934,E2 1244.934} C_VEL
LIN {X 0,Y 747.752,Z 1025.584,A -85,B 0,C 180,E1 1247.734,E2 1247.734} C_VEL
LIN {X 0,Y 747.988,Z 990.319,A -85,B 0,C 180,E1 1249.833,E2 1249.833} C_VEL
LIN {X 0,Y 748.13,Z 949.046,A -85,B 0,C 180,E1 1250.881,E2 1250.881} C_VEL
LIN {X 0,Y 747.604,Z 831.999,A -85,B 0,C 180,E1 1252.161,E2 1252.161} C_VEL
LIN {X 0,Y 747.841,Z 762.06,A -85,B 0,C 180,E1 1254.796,E2 1254.796} C_VEL
LIN {X 0,Y 746.34,Z 762.06,A -85,B 0,C 180,E1 1261.736,E2 1261.736} C_VEL
LIN {X 0,Y 739.339,Z 762.06,A -85,B 0,C 180,E1 1264.417,E2 1264.417} C_VEL
LIN {X 0,Y 739.197,Z 762.06,A -85,B 0,C 180,E1 1272.973,E2 1272.973} C_VEL
LIN {X 0,Y 739.009,Z 762.06,A -85,B 0,C 180,E1 1281.094,E2 1281.094} C_VEL
LIN {X 0,Y 738.998,Z 762.06,A -85,B 0,C 180,E1 1289.299,E2 1289.299} C_VEL
LIN {X 0,Y 738.685,Z 762.06,A -85,B 0,C 180,E1 1297.788,E2 1297.788} C_VEL
LIN {X 0,Y 738.766,Z 762.06,A -85,B 0,C 180,E1 1306.567,E2 1306.567} C_VEL
LIN {X 0,Y 738.99,Z 763.481,A -85,B 0,C 180,E1 1312.285,E2 1312.285} C_VEL
LIN {X 0,Y 743.824,Z 776.685,A -85,B 0,C 180,E1 1312.729,E2 1312.729} C_VEL
LIN {X 0,Y 743.938,Z 866.149,A -85,B 0,C 180,E1 1314.073,E2 1314.073} C_VEL
LIN {X 0,Y 743.052,Z 936.649,A -85,B 0,C 180,E1 1316.214,E2 1316.214} C_VEL
LIN {X 0,Y 741.772,Z 1008.112,A -85,B 0,C 180,E1 1319.645,E2 1319.645} C_VEL
LIN {X 0,Y 740.425,Z 1073.156,A -85,B 0,C 180,E1 1324.167,E2 1324.167} C_VEL
LIN {X 0,Y 739.463,Z 1125.017,A -85,B 0,C 180,E1 1329.19,E2 1329.19} C_VEL
LIN {X 0,Y 739.068,Z 1161.97,A -85,B 0,C 180,E1 1334.143,E2 1334.143} C_VEL
LIN {X 0,Y 738.947,Z 1188.829,A -85,B 0,C 180,E1 1339.382,E2 1339.382} C_VEL
LIN {X 0,Y 739.082,Z 1204.818,A -85,B 0,C 180,E1 1344.731,E2 1344.731} C_VEL
LIN {X 0,Y 739.588,Z 1209.852,A -85,B 0,C 180,E1 1349.443,E2 1349.443} C_VEL
LIN {X 0,Y 739.443,Z 1204.698,A -85,B 0,C 180,E1 1355.33,E2 1355.33} C_VEL
LIN {X 0,Y 739.32,Z 1184.687,A -85,B 0,C 180,E1 1361.575,E2 1361.575} C_VEL
LIN {X 0,Y 739.433,Z 1151.009,A -85,B 0,C 180,E1 1367.497,E2 1367.497} C_VEL
LIN {X 0,Y 740.147,Z 1103.333,A -85,B 0,C 180,E1 1373.1,E2 1373.1} C_VEL
LIN {X 0,Y 741.163,Z 1044.03,A -85,B 0,C 180,E1 1378.045,E2 1378.045} C_VEL
LIN {X 0,Y 742.396,Z 974.953,A -85,B 0,C 180,E1 1382.118,E2 1382.118} C_VEL
LIN {X 0,Y 743.521,Z 902.419,A -85,B 0,C 180,E1 1384.962,E2 1384.962} C_VEL
LIN {X 0,Y 744.032,Z 829.081,A -85,B 0,C 180,E1 1386.617,E2 1386.617} C_VEL
LIN {X 0,Y 742.409,Z 769.775,A -85,B 0,C 180,E1 1387.436,E2 1387.436} C_VEL
LIN {X 0,Y 738.809,Z 762.06,A -85,B 0,C 180,E1 1387.812,E2 1387.812} C_VEL
LIN {X 0,Y 738.746,Z 762.06,A -85,B 0,C 180,E1 1396.478,E2 1396.478} C_VEL
LIN {X 0,Y 738.882,Z 762.06,A -85,B 0,C 180,E1 1404.262,E2 1404.262} C_VEL
LIN {X 0,Y 738.93,Z 762.06,A -85,B 0,C 180,E1 1411.11,E2 1411.11} C_VEL
LIN {X 0,Y 738.574,Z 762.06,A -85,B 0,C 180,E1 1417.626,E2 1417.626} C_VEL
LIN {X 0,Y 738.926,Z 762.06,A -85,B 0,C 180,E1 1425.092,E2 1425.092} C_VEL
LIN {X 0,Y 739.188,Z 762.06,A -85,B 0,C 180,E1 1432.298,E2 1432.298} C_VEL
LIN {X 0,Y 738.849,Z 762.06,A -85,B 0,C 180,E1 1440.554,E2 1440.554} C_VEL
LIN {X 0,Y 739.036,Z 762.06,A -85,B 0,C 180,E1 1447.634,E2 1447.634} C_VEL
LIN {X 0,Y 739.303,Z 762.06,A -85,B 0,C 180,E1 1454.829,E2 1454.829} C_VEL
LIN {X 0,Y 738.797,Z 762.06,A -85,B 0,C 180,E1 1463.57,E2 1463.57} C_VEL
LIN {X 0,Y 738.602,Z 762.06,A -85,B 0,C 180,E1 1471.549,E2 1471.549} C_VEL
LIN {X 0,Y 738.717,Z 762.06,A -85,B 0,C 180,E1 1478.744,E2 1478.744} C_VEL
LIN {X 0,Y 738.797,Z 762.06,A -85,B 0,C 180,E1 1486.483,E2 1486.483} C_VEL
LIN {X 0,Y 739.385,Z 763.962,A -85,B 0,C 180,E1 1492.629,E2 1492.629} C_VEL
LIN {X 0,Y 743.965,Z 781.136,A -85,B 0,C 180,E1 1493.101,E2 1493.101} C_VEL
LIN {X 0,Y 743.556,Z 859.242,A -85,B 0,C 180,E1 1494.599,E2 1494.599} C_VEL
LIN {X 0,Y 742.586,Z 932.243,A -85,B 0,C 180,E1 1497.246,E2 1497.246} C_VEL
LIN {X 0,Y 741.256,Z 1002.208,A -85,B 0,C 180,E1 1501.1,E2 1501.1} C_VEL
LIN {X 0,Y 740.132,Z 1062.815,A -85,B 0,C 180,E1 1505.84,E2 1505.84} C_VEL
LIN {X 0,Y 739.491,Z 1109.861,A -85,B 0,C 180,E1 1510.952,E2 1510.952} C_VEL
LIN {X 0,Y 739.163,Z 1144.676,A -85,B 0,C 180,E1 1516.313,E2 1516.313} C_VEL
LIN {X 0,Y 739.338,Z 1167.264,A -85,B 0,C 180,E1 1521.709,E2 1521.709} C_VEL
LIN {X 0,Y 739.44,Z 1178.391,A -85,B 0,C 180,E1 1527.028,E2 1527.028} C_VEL
LIN {X 0,Y 739.516,Z 1178.363,A -85,B 0,C 180,E1 1532.909,E2 1532.909} C_VEL
LIN {X 0,Y 739.245,Z 1164.256,A -85,B 0,C 180,E1 1539.121,E2 1539.121} C_VEL
LIN {X 0,Y 739.391,Z 1136.68,A -85,B 0,C 180,E1 1545.02,E2 1545.02} C_VEL
LIN {X 0,Y 739.879,Z 1095.599,A -85,B 0,C 180,E1 1550.684,E2 1550.684} C_VEL
LIN {X 0,Y 740.764,Z 1040.481,A -85,B 0,C 180,E1 1556.002,E2 1556.002} C_VEL
LIN {X 0,Y 741.897,Z 976.072,A -85,B 0,C 180,E1 1560.424,E2 1560.424} C_VEL
LIN {X 0,Y 743.084,Z 903.864,A -85,B 0,C 180,E1 1563.847,E2 1563.847} C_VEL
LIN {X 0,Y 743.939,Z 829.538,A -85,B 0,C 180,E1 1566.027,E2 1566.027} C_VEL
LIN {X 0,Y 742.138,Z 768.681,A -85,B 0,C 180,E1 1567.063,E2 1567.063} C_VEL
LIN {X 0,Y 739.192,Z 762.06,A -85,B 0,C 180,E1 1567.413,E2 1567.413} C_VEL
LIN {X 0,Y 738.973,Z 762.06,A -85,B 0,C 180,E1 1573.418,E2 1573.418} C_VEL
LIN {X 0,Y 739.228,Z 762.06,A -85,B 0,C 180,E1 1581.288,E2 1581.288} C_VEL
LIN {X 0,Y 739.774,Z 763.943,A -85,B 0,C 180,E1 1587.118,E2 1587.118} C_VEL
LIN {X 0,Y 739.527,Z 841.706,A -85,B 0,C 180,E1 1589.864,E2 1589.864} C_VEL
LIN {X 0,Y 740.188,Z 968.832,A -85,B 0,C 180,E1 1591.28,E2 1591.28} C_VEL
LIN {X 0,Y 739.972,Z 1008.882,A -85,B 0,C 180,E1 1592.911,E2 1592.911} C_VEL
LIN {X 0,Y 739.668,Z 1039.462,A -85,B 0,C 180,E1 1595.509,E2 1595.509} C_VEL
LIN {X 0,Y 739.427,Z 1055.543,A -85,B 0,C 180,E1 1598.336,E2 1598.336} C_VEL
LIN {X 0,Y 739.496,Z 1059.725,A -85,B 0,C 180,E1 1601.493,E2 1601.493} C_VEL
LIN {X 0,Y 739.567,Z 1050.33,A -85,B 0,C 180,E1 1604.766,E2 1604.766} C_VEL
LIN {X 0,Y 739.872,Z 1027.958,A -85,B 0,C 180,E1 1607.601,E2 1607.601} C_VEL
LIN {X 0,Y 740.062,Z 993.79,A -85,B 0,C 180,E1 1609.778,E2 1609.778} C_VEL
LIN {X 0,Y 740.242,Z 953.327,A -85,B 0,C 180,E1 1610.932,E2 1610.932} C_VEL
LIN {X 0,Y 739.749,Z 831.506,A -85,B 0,C 180,E1 1612.299,E2 1612.299} C_VEL
LIN {X 0,Y 739.853,Z 762.06,A -85,B 0,C 180,E1 1614.887,E2 1614.887} C_VEL
LIN {X 0,Y 739.339,Z 762.06,A -85,B 0,C 180,E1 1624.417,E2 1624.417} C_VEL
LIN {X 0,Y 730.411,Z 762.06,A -85,B 0,C 180,E1 1627.095,E2 1627.095} C_VEL
LIN {X 0,Y 730.688,Z 762.06,A -85,B 0,C 180,E1 1633.851,E2 1633.851} C_VEL
LIN {X 0,Y 730.834,Z 762.06,A -85,B 0,C 180,E1 1641.341,E2 1641.341} C_VEL
LIN {X 0,Y 731.026,Z 762.06,A -85,B 0,C 180,E1 1649.232,E2 1649.232} C_VEL
LIN {X 0,Y 730.669,Z 762.06,A -85,B 0,C 180,E1 1657.82,E2 1657.82} C_VEL
LIN {X 0,Y 730.95,Z 762.06,A -85,B 0,C 180,E1 1665.984,E2 1665.984} C_VEL
LIN {X 0,Y 730.671,Z 763.281,A -85,B 0,C 180,E1 1671.776,E2 1671.776} C_VEL
LIN {X 0,Y 737.46,Z 779.034,A -85,B 0,C 180,E1 1672.38,E2 1672.38} C_VEL
LIN {X 0,Y 737.401,Z 867.444,A -85,B 0,C 180,E1 1673.735,E2 1673.735} C_VEL
LIN {X 0,Y 736.201,Z 937.682,A -85,B 0,C 180,E1 1675.9,E2 1675.9} C_VEL
LIN {X 0,Y 734.598,Z 1008.461,A -85,B 0,C 180,E1 1679.338,E2 1679.338} C_VEL
LIN {X 0,Y 732.895,Z 1073.701,A -85,B 0,C 180,E1 1683.928,E2 1683.928} C_VEL
LIN {X 0,Y 731.643,Z 1126.152,A -85,B 0,C 180,E1 1689.091,E2 1689.091} C_VEL
LIN {X 0,Y 731.156,Z 1162.648,A -85,B 0,C 180,E1 1694.073,E2 1694.073} C_VEL
LIN {X 0,Y 731.016,Z 1188.83,A -85,B 0,C 180,E1 1699.266,E2 1699.266} C_VEL
LIN {X 0,Y 731.105,Z 1204.818,A -85,B 0,C 180,E1 1704.673,E2 1704.673} C_VEL
LIN {X 0,Y 731.609,Z 1209.854,A -85,B 0,C 180,E1 1709.437,E2 1709.437} C_VEL
LIN {X 0,Y 731.4,Z 1204.699,A -85,B 0,C 180,E1 1715.388,E2 1715.388} C_VEL
LIN {X 0,Y 731.413,Z 1186.046,A -85,B 0,C 180,E1 1721.398,E2 1721.398} C_VEL
LIN {X 0,Y 731.583,Z 1152.928,A -85,B 0,C 180,E1 1727.421,E2 1727.421} C_VEL
LIN {X 0,Y 732.464,Z 1106.237,A -85,B 0,C 180,E1 1733.067,E2 1733.067} C_VEL
LIN {X 0,Y 733.731,Z 1047.545,A -85,B 0,C 180,E1 1738.098,E2 1738.098} C_VEL
LIN {X 0,Y 735.272,Z 979.051,A -85,B 0,C 180,E1 1742.255,E2 1742.255} C_VEL
LIN {X 0,Y 736.769,Z 906.554,A -85,B 0,C 180,E1 1745.196,E2 1745.196} C_VEL
LIN {X 0,Y 737.565,Z 833.221,A -85,B 0,C 180,E1 1746.927,E2 1746.927} C_VEL
LIN {X 0,Y 736.038,Z 772.947,A -85,B 0,C 180,E1 1747.779,E2 1747.779} C_VEL
LIN {X 0,Y 730.436,Z 762.06,A -85,B 0,C 180,E1 1748.438,E2 1748.438} C_VEL
LIN {X 0,Y 730.969,Z 762.06,A -85,B 0,C 180,E1 1755.896,E2 1755.896} C_VEL
LIN {X 0,Y 730.951,Z 762.06,A -85,B 0,C 180,E1 1763.687,E2 1763.687} C_VEL
LIN {X 0,Y 731.06,Z 762.06,A -85,B 0,C 180,E1 1770.769,E2 1770.769} C_VEL
LIN {X 0,Y 730.569,Z 762.06,A -85,B 0,C 180,E1 1777.635,E2 1777.635} C_VEL
LIN {X 0,Y 730.954,Z 762.06,A -85,B 0,C 180,E1 1784.975,E2 1784.975} C_VEL
LIN {X 0,Y 731.197,Z 762.06,A -85,B 0,C 180,E1 1792.213,E2 1792.213} C_VEL
LIN {X 0,Y 730.853,Z 762.06,A -85,B 0,C 180,E1 1800.56,E2 1800.56} C_VEL
LIN {X 0,Y 730.978,Z 762.06,A -85,B 0,C 180,E1 1807.719,E2 1807.719} C_VEL
LIN {X 0,Y 731.112,Z 762.06,A -85,B 0,C 180,E1 1815.072,E2 1815.072} C_VEL
LIN {X 0,Y 730.707,Z 762.06,A -85,B 0,C 180,E1 1823.847,E2 1823.847} C_VEL
LIN {X 0,Y 730.993,Z 762.06,A -85,B 0,C 180,E1 1830.525,E2 1830.525} C_VEL
LIN {X 0,Y 730.681,Z 762.06,A -85,B 0,C 180,E1 1838.806,E2 1838.806} C_VEL
LIN {X 0,Y 730.97,Z 762.06,A -85,B 0,C 180,E1 1845.898,E2 1845.898} C_VEL
LIN {X 0,Y 731.04,Z 763.983,A -85,B 0,C 180,E1 1852.129,E2 1852.129} C_VEL
LIN {X 0,Y 737.505,Z 778.756,A -85,B 0,C 180,E1 1852.695,E2 1852.695} C_VEL
LIN {X 0,Y 736.933,Z 857.877,A -85,B 0,C 180,E1 1854.194,E2 1854.194} C_VEL
LIN {X 0,Y 735.59,Z 932.91,A -85,B 0,C 180,E1 1856.927,E2 1856.927} C_VEL
LIN {X 0,Y 733.91,Z 1003.877,A -85,B 0,C 180,E1 1860.896,E2 1860.896} C_VEL
LIN {X 0,Y 732.473,Z 1064.362,A -85,B 0,C 180,E1 1865.713,E2 1865.713} C_VEL
LIN {X 0,Y 731.552,Z 1112.197,A -85,B 0,C 180,E1 1871.038,E2 1871.038} C_VEL
LIN {X 0,Y 731.064,Z 1146.755,A -85,B 0,C 180,E1 1876.567,E2 1876.567} C_VEL
LIN {X 0,Y 731.058,Z 1169.051,A -85,B 0,C 180,E1 1882.215,E2 1882.215} C_VEL
LIN {X 0,Y 731.444,Z 1178.391,A -85,B 0,C 180,E1 1886.996,E2 1886.996} C_VEL
LIN {X 0,Y 731.487,Z 1178.364,A -85,B 0,C 180,E1 1892.941,E2 1892.941} C_VEL
LIN {X 0,Y 731.356,Z 1165.277,A -85,B 0,C 180,E1 1898.92,E2 1898.92} C_VEL
LIN {X 0,Y 731.476,Z 1137.782,A -85,B 0,C 180,E1 1904.995,E2 1904.995} C_VEL
LIN {X 0,Y 732.061,Z 1096.953,A -85,B 0,C 180,E1 1910.757,E2 1910.757} C_VEL
LIN {X 0,Y 733.158,Z 1043.031,A -85,B 0,C 180,E1 1916.075,E2 1916.075} C_VEL
LIN {X 0,Y 734.69,Z 978.133,A -85,B 0,C 180,E1 1920.634,E2 1920.634} C_VEL
LIN {X 0,Y 736.26,Z 905.812,A -85,B 0,C 180,E1 1924.13,E2 1924.13} C_VEL
LIN {X 0,Y 737.402,Z 831.421,A -85,B 0,C 180,E1 1926.356,E2 1926.356} C_VEL
LIN {X 0,Y 735.8,Z 772.152,A -85,B 0,C 180,E1 1927.395,E2 1927.395} C_VEL
LIN {X 0,Y 730.993,Z 762.06,A -85,B 0,C 180,E1 1927.968,E2 1927.968} C_VEL
LIN {X 0,Y 730.5,Z 762.06,A -85,B 0,C 180,E1 1934.278,E2 1934.278} C_VEL
LIN {X 0,Y 730.842,Z 762.06,A -85,B 0,C 180,E1 1942.279,E2 1942.279} C_VEL
LIN {X 0,Y 731.785,Z 763.638,A -85,B 0,C 180,E1 1946.953,E2 1946.953} C_VEL
LIN {X 0,Y 731.676,Z 843.383,A -85,B 0,C 180,E1 1949.76,E2 1949.76} C_VEL
LIN {X 0,Y 732.33,Z 968.341,A -85,B 0,C 180,E1 1951.163,E2 1951.163} C_VEL
LIN {X 0,Y 732.01,Z 1008.343,A -85,B 0,C 180,E1 1952.791,E2 1952.791} C_VEL
LIN {X 0,Y 731.619,Z 1038.612,A -85,B 0,C 180,E1 1955.348,E2 1955.348} C_VEL
LIN {X 0,Y 731.462,Z 1055.924,A -85,B 0,C 180,E1 1958.434,E2 1958.434} C_VEL
LIN {X 0,Y 731.456,Z 1059.847,A -85,B 0,C 180,E1 1961.282,E2 1961.282} C_VEL
LIN {X 0,Y 731.473,Z 1051.486,A -85,B 0,C 180,E1 1964.585,E2 1964.585} C_VEL
LIN {X 0,Y 731.917,Z 1028.588,A -85,B 0,C 180,E1 1967.616,E2 1967.616} C_VEL
LIN {X 0,Y 732.171,Z 995.469,A -85,B 0,C 180,E1 1969.797,E2 1969.797} C_VEL
LIN {X 0,Y 732.387,Z 954.746,A -85,B 0,C 180,E1 1971.022,E2 1971.022} C_VEL
LIN {X 0,Y 731.895,Z 832.025,A -85,B 0,C 180,E1 1972.403,E2 1972.403} C_VEL
LIN {X 0,Y 731.82,Z 762.06,A -85,B 0,C 180,E1 1975.129,E2 1975.129} C_VEL
LIN {X 0,Y 731.281,Z 762.06,A -85,B 0,C 180,E1 1985.392,E2 1985.392} C_VEL
LIN {X 0,Y 730.411,Z 762.06,A -85,B 0,C 180,E1 1987.095,E2 1987.095} C_VEL
LIN {X 0,Y 722.393,Z 762.06,A -85,B 0,C 180,E1 1989.813,E2 1989.813} C_VEL
LIN {X 0,Y 722.204,Z 762.06,A -85,B 0,C 180,E1 1995.261,E2 1995.261} C_VEL
LIN {X 0,Y 722.699,Z 762.06,A -85,B 0,C 180,E1 2001.593,E2 2001.593} C_VEL
LIN {X 0,Y 722.841,Z 762.06,A -85,B 0,C 180,E1 2009.596,E2 2009.596} C_VEL
LIN {X 0,Y 722.523,Z 762.06,A -85,B 0,C 180,E1 2018.098,E2 2018.098} C_VEL
LIN {X 0,Y 722.7,Z 762.06,A -85,B 0,C 180,E1 2026.462,E2 2026.462} C_VEL
LIN {X 0,Y 722.532,Z 763.931,A -85,B 0,C 180,E1 2031.274,E2 2031.274} C_VEL
LIN {X 0,Y 731.109,Z 781.802,A -85,B 0,C 180,E1 2032.03,E2 2032.03} C_VEL
LIN {X 0,Y 730.867,Z 868.437,A -85,B 0,C 180,E1 2033.382,E2 2033.382} C_VEL
LIN {X 0,Y 729.38,Z 938.569,A -85,B 0,C 180,E1 2035.574,E2 2035.574} C_VEL
LIN {X 0,Y 727.354,Z 1010.056,A -85,B 0,C 180,E1 2039.1,E2 2039.1} C_VEL
LIN {X 0,Y 725.333,Z 1074.189,A -85,B 0,C 180,E1 2043.677,E2 2043.677} C_VEL
LIN {X 0,Y 723.961,Z 1125.642,A -85,B 0,C 180,E1 2048.797,E2 2048.797} C_VEL
LIN {X 0,Y 723.275,Z 1162.646,A -85,B 0,C 180,E1 2053.894,E2 2053.894} C_VEL
LIN {X 0,Y 723.082,Z 1188.83,A -85,B 0,C 180,E1 2059.146,E2 2059.146} C_VEL
LIN {X 0,Y 723.137,Z 1204.819,A -85,B 0,C 180,E1 2064.614,E2 2064.614} C_VEL
LIN {X 0,Y 723.604,Z 1209.855,A -85,B 0,C 180,E1 2069.431,E2 2069.431} C_VEL
LIN {X 0,Y 723.39,Z 1204.699,A -85,B 0,C 180,E1 2075.448,E2 2075.448} C_VEL
LIN {X 0,Y 723.268,Z 1185.024,A -85,B 0,C 180,E1 2081.76,E2 2081.76} C_VEL
LIN {X 0,Y 723.543,Z 1152.121,A -85,B 0,C 180,E1 2087.736,E2 2087.736} C_VEL
LIN {X 0,Y 724.675,Z 1105.984,A -85,B 0,C 180,E1 2093.356,E2 2093.356} C_VEL
LIN {X 0,Y 726.308,Z 1046.799,A -85,B 0,C 180,E1 2098.467,E2 2098.467} C_VEL
LIN {X 0,Y 728.323,Z 977.777,A -85,B 0,C 180,E1 2102.668,E2 2102.668} C_VEL
LIN {X 0,Y 730.114,Z 906.563,A -85,B 0,C 180,E1 2105.565,E2 2105.565} C_VEL
LIN {X 0,Y 731.18,Z 832.224,A -85,B 0,C 180,E1 2107.32,E2 2107.32} C_VEL
LIN {X 0,Y 729.778,Z 776.549,A -85,B 0,C 180,E1 2108.116,E2 2108.116} C_VEL
LIN {X 0,Y 722.207,Z 762.06,A -85,B 0,C 180,E1 2108.959,E2 2108.959} C_VEL
LIN {X 0,Y 722.673,Z 762.06,A -85,B 0,C 180,E1 2116.463,E2 2116.463} C_VEL
LIN {X 0,Y 722.662,Z 762.06,A -85,B 0,C 180,E1 2124.691,E2 2124.691} C_VEL
LIN {X 0,Y 722.796,Z 762.06,A -85,B 0,C 180,E1 2131.776,E2 2131.776} C_VEL
LIN {X 0,Y 722.242,Z 762.06,A -85,B 0,C 180,E1 2138.392,E2 2138.392} C_VEL
LIN {X 0,Y 723.006,Z 762.06,A -85,B 0,C 180,E1 2144.756,E2 2144.756} C_VEL
LIN {X 0,Y 723.224,Z 762.06,A -85,B 0,C 180,E1 2152.127,E2 2152.127} C_VEL
LIN {X 0,Y 722.844,Z 762.06,A -85,B 0,C 180,E1 2160.566,E2 2160.566} C_VEL
LIN {X 0,Y 722.953,Z 762.06,A -85,B 0,C 180,E1 2167.805,E2 2167.805} C_VEL
LIN {X 0,Y 723.056,Z 762.06,A -85,B 0,C 180,E1 2175.17,E2 2175.17} C_VEL
LIN {X 0,Y 722.665,Z 762.06,A -85,B 0,C 180,E1 2183.95,E2 2183.95} C_VEL
LIN {X 0,Y 722.513,Z 762.06,A -85,B 0,C 180,E1 2191.67,E2 2191.67} C_VEL
LIN {X 0,Y 722.861,Z 762.06,A -85,B 0,C 180,E1 2198.212,E2 2198.212} C_VEL
LIN {X 0,Y 722.726,Z 762.06,A -85,B 0,C 180,E1 2206.357,E2 2206.357} C_VEL
LIN {X 0,Y 722.744,Z 763.907,A -85,B 0,C 180,E1 2211.616,E2 2211.616} C_VEL
LIN {X 0,Y 731.167,Z 781.872,A -85,B 0,C 180,E1 2212.354,E2 2212.354} C_VEL
LIN {X 0,Y 730.3,Z 860.709,A -85,B 0,C 180,E1 2213.901,E2 2213.901} C_VEL
LIN {X 0,Y 728.622,Z 934.045,A -85,B 0,C 180,E1 2216.623,E2 2216.623} C_VEL
LIN {X 0,Y 726.61,Z 1003.874,A -85,B 0,C 180,E1 2220.575,E2 2220.575} C_VEL
LIN {X 0,Y 724.859,Z 1064.917,A -85,B 0,C 180,E1 2225.493,E2 2225.493} C_VEL
LIN {X 0,Y 723.665,Z 1113.558,A -85,B 0,C 180,E1 2231.001,E2 2231.001} C_VEL
LIN {X 0,Y 723.073,Z 1147.787,A -85,B 0,C 180,E1 2236.621,E2 2236.621} C_VEL
LIN {X 0,Y 723.097,Z 1169.05,A -85,B 0,C 180,E1 2242.128,E2 2242.128} C_VEL
LIN {X 0,Y 723.44,Z 1178.391,A -85,B 0,C 180,E1 2246.962,E2 2246.962} C_VEL
LIN {X 0,Y 723.458,Z 1178.365,A -85,B 0,C 180,E1 2252.974,E2 2252.974} C_VEL
LIN {X 0,Y 723.324,Z 1165.279,A -85,B 0,C 180,E1 2259.02,E2 2259.02} C_VEL
LIN {X 0,Y 723.477,Z 1137.785,A -85,B 0,C 180,E1 2265.165,E2 2265.165} C_VEL
LIN {X 0,Y 724.212,Z 1096.725,A -85,B 0,C 180,E1 2271.02,E2 2271.02} C_VEL
LIN {X 0,Y 725.657,Z 1043.038,A -85,B 0,C 180,E1 2276.365,E2 2276.365} C_VEL
LIN {X 0,Y 727.52,Z 978.142,A -85,B 0,C 180,E1 2280.969,E2 2280.969} C_VEL
LIN {X 0,Y 729.421,Z 907.201,A -85,B 0,C 180,E1 2284.436,E2 2284.436} C_VEL
LIN {X 0,Y 730.889,Z 833.764,A -85,B 0,C 180,E1 2286.681,E2 2286.681} C_VEL
LIN {X 0,Y 729.561,Z 775.676,A -85,B 0,C 180,E1 2287.729,E2 2287.729} C_VEL
LIN {X 0,Y 722.934,Z 762.06,A -85,B 0,C 180,E1 2288.359,E2 2288.359} C_VEL
LIN {X 0,Y 722.179,Z 762.06,A -85,B 0,C 180,E1 2295.316,E2 2295.316} C_VEL
LIN {X 0,Y 722.98,Z 762.06,A -85,B 0,C 180,E1 2301.856,E2 2301.856} C_VEL
LIN {X 0,Y 723.756,Z 763.317,A -85,B 0,C 180,E1 2306.782,E2 2306.782} C_VEL
LIN {X 0,Y 723.847,Z 840.208,A -85,B 0,C 180,E1 2309.606,E2 2309.606} C_VEL
LIN {X 0,Y 724.422,Z 969.435,A -85,B 0,C 180,E1 2311.085,E2 2311.085} C_VEL
LIN {X 0,Y 724.088,Z 1008.773,A -85,B 0,C 180,E1 2312.729,E2 2312.729} C_VEL
LIN {X 0,Y 723.628,Z 1038.771,A -85,B 0,C 180,E1 2315.303,E2 2315.303} C_VEL
LIN {X 0,Y 723.501,Z 1056.22,A -85,B 0,C 180,E1 2318.508,E2 2318.508} C_VEL
LIN {X 0,Y 723.454,Z 1059.967,A -85,B 0,C 180,E1 2321.067,E2 2321.067} C_VEL
LIN {X 0,Y 723.489,Z 1051.479,A -85,B 0,C 180,E1 2324.625,E2 2324.625} C_VEL
LIN {X 0,Y 723.955,Z 1029.205,A -85,B 0,C 180,E1 2327.631,E2 2327.631} C_VEL
LIN {X 0,Y 724.249,Z 994.714,A -85,B 0,C 180,E1 2329.931,E2 2329.931} C_VEL
LIN {X 0,Y 724.531,Z 953.38,A -85,B 0,C 180,E1 2331.151,E2 2331.151} C_VEL
LIN {X 0,Y 724.036,Z 832.549,A -85,B 0,C 180,E1 2332.51,E2 2332.51} C_VEL
LIN {X 0,Y 723.816,Z 762.06,A -85,B 0,C 180,E1 2335.226,E2 2335.226} C_VEL
LIN {X 0,Y 723.244,Z 762.06,A -85,B 0,C 180,E1 2345.452,E2 2345.452} C_VEL
LIN {X 0,Y 722.393,Z 762.06,A -85,B 0,C 180,E1 2349.813,E2 2349.813} C_VEL
LIN {X 0,Y 715.174,Z 762.06,A -85,B 0,C 180,E1 2352.596,E2 2352.596} C_VEL
LIN {X 0,Y 715.01,Z 762.06,A -85,B 0,C 180,E1 2360.533,E2 2360.533} C_VEL
LIN {X 0,Y 714.634,Z 762.06,A -85,B 0,C 180,E1 2369.971,E2 2369.971} C_VEL
LIN {X 0,Y 714.716,Z 762.06,A -85,B 0,C 180,E1 2377.292,E2 2377.292} C_VEL
LIN {X 0,Y 714.721,Z 762.06,A -85,B 0,C 180,E1 2386.417,E2 2386.417} C_VEL
LIN {X 0,Y 714.22,Z 763.197,A -85,B 0,C 180,E1 2390.728,E2 2390.728} C_VEL
LIN {X 0,Y 724.788,Z 784.102,A -85,B 0,C 180,E1 2391.667,E2 2391.667} C_VEL
LIN {X 0,Y 724.356,Z 869.401,A -85,B 0,C 180,E1 2393.023,E2 2393.023} C_VEL
LIN {X 0,Y 722.58,Z 939.802,A -85,B 0,C 180,E1 2395.256,E2 2395.256} C_VEL
LIN {X 0,Y 720.152,Z 1010.723,A -85,B 0,C 180,E1 2398.798,E2 2398.798} C_VEL
LIN {X 0,Y 717.785,Z 1075.046,A -85,B 0,C 180,E1 2403.454,E2 2403.454} C_VEL
LIN {X 0,Y 716.154,Z 1127.078,A -85,B 0,C 180,E1 2408.728,E2 2408.728} C_VEL
LIN {X 0,Y 715.282,Z 1164.516,A -85,B 0,C 180,E1 2414.026,E2 2414.026} C_VEL
LIN {X 0,Y 715.013,Z 1190.034,A -85,B 0,C 180,E1 2419.332,E2 2419.332} C_VEL
LIN {X 0,Y 715.161,Z 1204.819,A -85,B 0,C 180,E1 2424.554,E2 2424.554} C_VEL
LIN {X 0,Y 714.98,Z 1209.839,A -85,B 0,C 180,E1 2430.64,E2 2430.64} C_VEL
LIN {X 0,Y 715.036,Z 1203.45,A -85,B 0,C 180,E1 2436.123,E2 2436.123} C_VEL
LIN {X 0,Y 715.364,Z 1186.052,A -85,B 0,C 180,E1 2441.658,E2 2441.658} C_VEL
LIN {X 0,Y 715.701,Z 1153.744,A -85,B 0,C 180,E1 2447.698,E2 2447.698} C_VEL
LIN {X 0,Y 716.965,Z 1108.007,A -85,B 0,C 180,E1 2453.414,E2 2453.414} C_VEL
LIN {X 0,Y 718.886,Z 1048.871,A -85,B 0,C 180,E1 2458.633,E2 2458.633} C_VEL
LIN {X 0,Y 721.268,Z 980.408,A -85,B 0,C 180,E1 2462.889,E2 2462.889} C_VEL
LIN {X 0,Y 723.455,Z 908.52,A -85,B 0,C 180,E1 2465.878,E2 2465.878} C_VEL
LIN {X 0,Y 724.751,Z 835.507,A -85,B 0,C 180,E1 2467.656,E2 2467.656} C_VEL
LIN {X 0,Y 723.283,Z 779.323,A -85,B 0,C 180,E1 2468.487,E2 2468.487} C_VEL
LIN {X 0,Y 714.06,Z 762.06,A -85,B 0,C 180,E1 2469.433,E2 2469.433} C_VEL
LIN {X 0,Y 714.706,Z 762.06,A -85,B 0,C 180,E1 2476.325,E2 2476.325} C_VEL
LIN {X 0,Y 714.613,Z 762.06,A -85,B 0,C 180,E1 2484.888,E2 2484.888} C_VEL
LIN {X 0,Y 714.813,Z 762.06,A -85,B 0,C 180,E1 2491.822,E2 2491.822} C_VEL
LIN {X 0,Y 714.315,Z 762.06,A -85,B 0,C 180,E1 2498.14,E2 2498.14} C_VEL
LIN {X 0,Y 714.832,Z 762.06,A -85,B 0,C 180,E1 2505.098,E2 2505.098} C_VEL
LIN {X 0,Y 715.219,Z 762.06,A -85,B 0,C 180,E1 2512.038,E2 2512.038} C_VEL
LIN {X 0,Y 714.85,Z 762.06,A -85,B 0,C 180,E1 2520.572,E2 2520.572} C_VEL
LIN {X 0,Y 714.897,Z 762.06,A -85,B 0,C 180,E1 2527.893,E2 2527.893} C_VEL
LIN {X 0,Y 714.955,Z 762.06,A -85,B 0,C 180,E1 2535.346,E2 2535.346} C_VEL
LIN {X 0,Y 714.935,Z 762.06,A -85,B 0,C 180,E1 2543.078,E2 2543.078} C_VEL
LIN {X 0,Y 714.632,Z 762.06,A -85,B 0,C 180,E1 2551.302,E2 2551.302} C_VEL
LIN {X 0,Y 714.47,Z 762.06,A -85,B 0,C 180,E1 2559.13,E2 2559.13} C_VEL
LIN {X 0,Y 714.738,Z 762.06,A -85,B 0,C 180,E1 2566.329,E2 2566.329} C_VEL
LIN {X 0,Y 714.519,Z 763.955,A -85,B 0,C 180,E1 2571.093,E2 2571.093} C_VEL
LIN {X 0,Y 724.854,Z 784.686,A -85,B 0,C 180,E1 2572.004,E2 2572.004} C_VEL
LIN {X 0,Y 723.713,Z 862.736,A -85,B 0,C 180,E1 2573.581,E2 2573.581} C_VEL
LIN {X 0,Y 721.662,Z 936.112,A -85,B 0,C 180,E1 2576.358,E2 2576.358} C_VEL
LIN {X 0,Y 719.271,Z 1005.69,A -85,B 0,C 180,E1 2580.37,E2 2580.37} C_VEL
LIN {X 0,Y 717.143,Z 1066.842,A -85,B 0,C 180,E1 2585.405,E2 2585.405} C_VEL
LIN {X 0,Y 715.802,Z 1114.676,A -85,B 0,C 180,E1 2590.945,E2 2590.945} C_VEL
LIN {X 0,Y 715.158,Z 1147.786,A -85,B 0,C 180,E1 2596.47,E2 2596.47} C_VEL
LIN {X 0,Y 715.137,Z 1169.05,A -85,B 0,C 180,E1 2602.04,E2 2602.04} C_VEL
LIN {X 0,Y 715.436,Z 1178.391,A -85,B 0,C 180,E1 2606.928,E2 2606.928} C_VEL
LIN {X 0,Y 715.43,Z 1178.366,A -85,B 0,C 180,E1 2613.007,E2 2613.007} C_VEL
LIN {X 0,Y 715.279,Z 1165.282,A -85,B 0,C 180,E1 2619.122,E2 2619.122} C_VEL
LIN {X 0,Y 715.607,Z 1139.554,A -85,B 0,C 180,E1 2625.021,E2 2625.021} C_VEL
LIN {X 0,Y 716.409,Z 1098.422,A -85,B 0,C 180,E1 2631.056,E2 2631.056} C_VEL
LIN {X 0,Y 718.117,Z 1043.484,A -85,B 0,C 180,E1 2636.626,E2 2636.626} C_VEL
LIN {X 0,Y 720.329,Z 978.813,A -85,B 0,C 180,E1 2641.272,E2 2641.272} C_VEL
LIN {X 0,Y 722.671,Z 907.228,A -85,B 0,C 180,E1 2644.804,E2 2644.804} C_VEL
LIN {X 0,Y 724.436,Z 833.769,A -85,B 0,C 180,E1 2647.062,E2 2647.062} C_VEL
LIN {X 0,Y 723.394,Z 778.928,A -85,B 0,C 180,E1 2648.068,E2 2648.068} C_VEL
LIN {X 0,Y 714.883,Z 762.06,A -85,B 0,C 180,E1 2648.919,E2 2648.919} C_VEL
LIN {X 0,Y 714.176,Z 762.06,A -85,B 0,C 180,E1 2655.331,E2 2655.331} C_VEL
LIN {X 0,Y 714.734,Z 762.06,A -85,B 0,C 180,E1 2662.816,E2 2662.816} C_VEL
LIN {X 0,Y 715.748,Z 763.611,A -85,B 0,C 180,E1 2666.632,E2 2666.632} C_VEL
LIN {X 0,Y 716.015,Z 840.965,A -85,B 0,C 180,E1 2669.488,E2 2669.488} C_VEL
LIN {X 0,Y 716.558,Z 969.693,A -85,B 0,C 180,E1 2670.983,E2 2670.983} C_VEL
LIN {X 0,Y 716.159,Z 1009.409,A -85,B 0,C 180,E1 2672.679,E2 2672.679} C_VEL
LIN {X 0,Y 715.602,Z 1038.183,A -85,B 0,C 180,E1 2675.167,E2 2675.167} C_VEL
LIN {X 0,Y 715.409,Z 1055.56,A -85,B 0,C 180,E1 2678.252,E2 2678.252} C_VEL
LIN {X 0,Y 715.441,Z 1059.97,A -85,B 0,C 180,E1 2680.847,E2 2680.847} C_VEL
LIN {X 0,Y 715.404,Z 1052.754,A -85,B 0,C 180,E1 2684.38,E2 2684.38} C_VEL
LIN {X 0,Y 716.01,Z 1031.369,A -85,B 0,C 180,E1 2687.492,E2 2687.492} C_VEL
LIN {X 0,Y 716.298,Z 997.84,A -85,B 0,C 180,E1 2689.882,E2 2689.882} C_VEL
LIN {X 0,Y 716.627,Z 956.961,A -85,B 0,C 180,E1 2691.206,E2 2691.206} C_VEL
LIN {X 0,Y 716.156,Z 832.082,A -85,B 0,C 180,E1 2692.656,E2 2692.656} C_VEL
LIN {X 0,Y 715.806,Z 762.06,A -85,B 0,C 180,E1 2695.477,E2 2695.477} C_VEL
LIN {X 0,Y 715.194,Z 762.06,A -85,B 0,C 180,E1 2705.514,E2 2705.514} C_VEL
LIN {X 0,Y 715.174,Z 762.06,A -85,B 0,C 180,E1 2712.596,E2 2712.596} C_VEL
LIN {X 0,Y 706.192,Z 762.06,A -85,B 0,C 180,E1 2715.37,E2 2715.37} C_VEL
LIN {X 0,Y 706.442,Z 762.06,A -85,B 0,C 180,E1 2722.116,E2 2722.116} C_VEL
LIN {X 0,Y 706.69,Z 762.06,A -85,B 0,C 180,E1 2729.657,E2 2729.657} C_VEL
LIN {X 0,Y 706.512,Z 762.06,A -85,B 0,C 180,E1 2737.783,E2 2737.783} C_VEL
LIN {X 0,Y 706.787,Z 762.06,A -85,B 0,C 180,E1 2746.035,E2 2746.035} C_VEL
LIN {X 0,Y 706.141,Z 763.292,A -85,B 0,C 180,E1 2750.191,E2 2750.191} C_VEL
LIN {X 0,Y 718.507,Z 787.486,A -85,B 0,C 180,E1 2751.312,E2 2751.312} C_VEL
LIN {X 0,Y 717.868,Z 870.32,A -85,B 0,C 180,E1 2752.655,E2 2752.655} C_VEL
LIN {X 0,Y 715.758,Z 941.699,A -85,B 0,C 180,E1 2754.959,E2 2754.959} C_VEL
LIN {X 0,Y 713.002,Z 1011.255,A -85,B 0,C 180,E1 2758.484,E2 2758.484} C_VEL
LIN {X 0,Y 710.303,Z 1075.719,A -85,B 0,C 180,E1 2763.211,E2 2763.211} C_VEL
LIN {X 0,Y 708.426,Z 1127.093,A -85,B 0,C 180,E1 2768.486,E2 2768.486} C_VEL
LIN {X 0,Y 707.418,Z 1164.516,A -85,B 0,C 180,E1 2773.843,E2 2773.843} C_VEL
LIN {X 0,Y 706.956,Z 1191.179,A -85,B 0,C 180,E1 2779.522,E2 2779.522} C_VEL
LIN {X 0,Y 706.955,Z 1205.925,A -85,B 0,C 180,E1 2785.108,E2 2785.108} C_VEL
LIN {X 0,Y 706.975,Z 1209.841,A -85,B 0,C 180,E1 2790.648,E2 2790.648} C_VEL
LIN {X 0,Y 707.029,Z 1203.45,A -85,B 0,C 180,E1 2796.193,E2 2796.193} C_VEL
LIN {X 0,Y 707.186,Z 1184.902,A -85,B 0,C 180,E1 2802.062,E2 2802.062} C_VEL
LIN {X 0,Y 707.763,Z 1153.711,A -85,B 0,C 180,E1 2807.908,E2 2807.908} C_VEL
LIN {X 0,Y 709.256,Z 1108.325,A -85,B 0,C 180,E1 2813.651,E2 2813.651} C_VEL
LIN {X 0,Y 711.523,Z 1048.877,A -85,B 0,C 180,E1 2818.957,E2 2818.957} C_VEL
LIN {X 0,Y 714.326,Z 980.173,A -85,B 0,C 180,E1 2823.262,E2 2823.262} C_VEL
LIN {X 0,Y 716.849,Z 908.529,A -85,B 0,C 180,E1 2826.261,E2 2826.261} C_VEL
LIN {X 0,Y 718.435,Z 834.817,A -85,B 0,C 180,E1 2828.057,E2 2828.057} C_VEL
LIN {X 0,Y 717.097,Z 782.86,A -85,B 0,C 180,E1 2828.836,E2 2828.836} C_VEL
LIN {X 0,Y 705.977,Z 762.06,A -85,B 0,C 180,E1 2829.955,E2 2829.955} C_VEL
LIN {X 0,Y 706.785,Z 762.06,A -85,B 0,C 180,E1 2836.034,E2 2836.034} C_VEL
LIN {X 0,Y 706.788,Z 762.06,A -85,B 0,C 180,E1 2843.774,E2 2843.774} C_VEL
LIN {X 0,Y 706.885,Z 762.06,A -85,B 0,C 180,E1 2851.081,E2 2851.081} C_VEL
LIN {X 0,Y 706.404,Z 762.06,A -85,B 0,C 180,E1 2857.883,E2 2857.883} C_VEL
LIN {X 0,Y 706.58,Z 762.06,A -85,B 0,C 180,E1 2865.666,E2 2865.666} C_VEL
LIN {X 0,Y 706.706,Z 762.06,A -85,B 0,C 180,E1 2873.182,E2 2873.182} C_VEL
LIN {X 0,Y 706.841,Z 762.06,A -85,B 0,C 180,E1 2880.579,E2 2880.579} C_VEL
LIN {X 0,Y 706.846,Z 762.06,A -85,B 0,C 180,E1 2887.984,E2 2887.984} C_VEL
LIN {X 0,Y 706.834,Z 762.06,A -85,B 0,C 180,E1 2895.527,E2 2895.527} C_VEL
LIN {X 0,Y 706.6,Z 762.06,A -85,B 0,C 180,E1 2904.048,E2 2904.048} C_VEL
LIN {X 0,Y 706.418,Z 762.06,A -85,B 0,C 180,E1 2911.897,E2 2911.897} C_VEL
LIN {X 0,Y 706.434,Z 762.06,A -85,B 0,C 180,E1 2919.269,E2 2919.269} C_VEL
LIN {X 0,Y 706.84,Z 762.06,A -85,B 0,C 180,E1 2925.927,E2 2925.927} C_VEL
LIN {X 0,Y 706.343,Z 763.888,A -85,B 0,C 180,E1 2930.555,E2 2930.555} C_VEL
LIN {X 0,Y 718.576,Z 788.733,A -85,B 0,C 180,E1 2931.666,E2 2931.666} C_VEL
LIN {X 0,Y 717.155,Z 865.998,A -85,B 0,C 180,E1 2933.293,E2 2933.293} C_VEL
LIN {X 0,Y 714.707,Z 939.955,A -85,B 0,C 180,E1 2936.177,E2 2936.177} C_VEL
LIN {X 0,Y 711.812,Z 1009.909,A -85,B 0,C 180,E1 2940.333,E2 2940.333} C_VEL
LIN {X 0,Y 709.343,Z 1070.367,A -85,B 0,C 180,E1 2945.48,E2 2945.48} C_VEL
LIN {X 0,Y 707.824,Z 1116.885,A -85,B 0,C 180,E1 2951.047,E2 2951.047} C_VEL
LIN {X 0,Y 707.137,Z 1149.334,A -85,B 0,C 180,E1 2956.63,E2 2956.63} C_VEL
LIN {X 0,Y 707.209,Z 1169.049,A -85,B 0,C 180,E1 2961.951,E2 2961.951} C_VEL
LIN {X 0,Y 707.431,Z 1178.391,A -85,B 0,C 180,E1 2966.894,E2 2966.894} C_VEL
LIN {X 0,Y 707.403,Z 1178.367,A -85,B 0,C 180,E1 2973.041,E2 2973.041} C_VEL
LIN {X 0,Y 707.259,Z 1165.284,A -85,B 0,C 180,E1 2979.226,E2 2979.226} C_VEL
LIN {X 0,Y 707.616,Z 1139.659,A -85,B 0,C 180,E1 2985.177,E2 2985.177} C_VEL
LIN {X 0,Y 708.587,Z 1099.342,A -85,B 0,C 180,E1 2991.188,E2 2991.188} C_VEL
LIN {X 0,Y 710.555,Z 1045.202,A -85,B 0,C 180,E1 2996.78,E2 2996.78} C_VEL
LIN {X 0,Y 713.094,Z 981.328,A -85,B 0,C 180,E1 3001.463,E2 3001.463} C_VEL
LIN {X 0,Y 715.787,Z 910.763,A -85,B 0,C 180,E1 3005.034,E2 3005.034} C_VEL
LIN {X 0,Y 717.902,Z 837.224,A -85,B 0,C 180,E1 3007.372,E2 3007.372} C_VEL
LIN {X 0,Y 717.006,Z 782.09,A -85,B 0,C 180,E1 3008.43,E2 3008.43} C_VEL
LIN {X 0,Y 706.872,Z 762.06,A -85,B 0,C 180,E1 3009.516,E2 3009.516} C_VEL
LIN {X 0,Y 706.11,Z 762.06,A -85,B 0,C 180,E1 3015.997,E2 3015.997} C_VEL
LIN {X 0,Y 706.78,Z 762.06,A -85,B 0,C 180,E1 3022.325,E2 3022.325} C_VEL
LIN {X 0,Y 707.7,Z 763.79,A -85,B 0,C 180,E1 3026.468,E2 3026.468} C_VEL
LIN {X 0,Y 708.176,Z 842.649,A -85,B 0,C 180,E1 3029.376,E2 3029.376} C_VEL
LIN {X 0,Y 708.684,Z 968.523,A -85,B 0,C 180,E1 3030.84,E2 3030.84} C_VEL
LIN {X 0,Y 708.186,Z 1008.483,A -85,B 0,C 180,E1 3032.527,E2 3032.527} C_VEL
LIN {X 0,Y 707.643,Z 1038.634,A -85,B 0,C 180,E1 3035.159,E2 3035.159} C_VEL
LIN {X 0,Y 707.492,Z 1056.155,A -85,B 0,C 180,E1 3038.426,E2 3038.426} C_VEL
LIN {X 0,Y 707.533,Z 1059.446,A -85,B 0,C 180,E1 3041.922,E2 3041.922} C_VEL
LIN {X 0,Y 707.872,Z 1047.529,A -85,B 0,C 180,E1 3045.464,E2 3045.464} C_VEL
LIN {X 0,Y 707.856,Z 1021.775,A -85,B 0,C 180,E1 3048.444,E2 3048.444} C_VEL
LIN {X 0,Y 708.433,Z 985.809,A -85,B 0,C 180,E1 3050.519,E2 3050.519} C_VEL
LIN {X 0,Y 708.806,Z 944.234,A -85,B 0,C 180,E1 3051.496,E2 3051.496} C_VEL
LIN {X 0,Y 708.31,Z 831.595,A -85,B 0,C 180,E1 3052.807,E2 3052.807} C_VEL
LIN {X 0,Y 707.791,Z 762.06,A -85,B 0,C 180,E1 3055.579,E2 3055.579} C_VEL
LIN {X 0,Y 707.155,Z 762.06,A -85,B 0,C 180,E1 3065.577,E2 3065.577} C_VEL
LIN {X 0,Y 707.114,Z 762.06,A -85,B 0,C 180,E1 3073.057,E2 3073.057} C_VEL
LIN {X 0,Y 706.192,Z 762.06,A -85,B 0,C 180,E1 3075.37,E2 3075.37} C_VEL
LIN {X 0,Y 698.483,Z 762.06,A -85,B 0,C 180,E1 3078.199,E2 3078.199} C_VEL
LIN {X 0,Y 698.118,Z 762.06,A -85,B 0,C 180,E1 3085.656,E2 3085.656} C_VEL
LIN {X 0,Y 698.043,Z 762.06,A -85,B 0,C 180,E1 3092.219,E2 3092.219} C_VEL
LIN {X 0,Y 698.307,Z 762.06,A -85,B 0,C 180,E1 3098.307,E2 3098.307} C_VEL
LIN {X 0,Y 698.44,Z 762.06,A -85,B 0,C 180,E1 3106.863,E2 3106.863} C_VEL
LIN {X 0,Y 698.078,Z 763.444,A -85,B 0,C 180,E1 3109.639,E2 3109.639} C_VEL
LIN {X 0,Y 712.216,Z 792.174,A -85,B 0,C 180,E1 3110.966,E2 3110.966} C_VEL
LIN {X 0,Y 711.419,Z 873.376,A -85,B 0,C 180,E1 3112.338,E2 3112.338} C_VEL
LIN {X 0,Y 708.944,Z 944.299,A -85,B 0,C 180,E1 3114.687,E2 3114.687} C_VEL
LIN {X 0,Y 705.759,Z 1014.632,A -85,B 0,C 180,E1 3118.344,E2 3118.344} C_VEL
LIN {X 0,Y 702.736,Z 1077.649,A -85,B 0,C 180,E1 3123.073,E2 3123.073} C_VEL
LIN {X 0,Y 700.632,Z 1128.313,A -85,B 0,C 180,E1 3128.386,E2 3128.386} C_VEL
LIN {X 0,Y 699.553,Z 1164.516,A -85,B 0,C 180,E1 3133.657,E2 3133.657} C_VEL
LIN {X 0,Y 699.012,Z 1191.18,A -85,B 0,C 180,E1 3139.401,E2 3139.401} C_VEL
LIN {X 0,Y 698.992,Z 1205.924,A -85,B 0,C 180,E1 3145.052,E2 3145.052} C_VEL
LIN {X 0,Y 698.987,Z 1209.843,A -85,B 0,C 180,E1 3150.655,E2 3150.655} C_VEL
LIN {X 0,Y 699.028,Z 1203.451,A -85,B 0,C 180,E1 3156.264,E2 3156.264} C_VEL
LIN {X 0,Y 699.268,Z 1186.057,A -85,B 0,C 180,E1 3161.93,E2 3161.93} C_VEL
LIN {X 0,Y 699.86,Z 1154.677,A -85,B 0,C 180,E1 3167.968,E2 3167.968} C_VEL
LIN {X 0,Y 701.534,Z 1108.612,A -85,B 0,C 180,E1 3173.897,E2 3173.897} C_VEL
LIN {X 0,Y 704.121,Z 1050.683,A -85,B 0,C 180,E1 3179.152,E2 3179.152} C_VEL
LIN {X 0,Y 707.31,Z 982.784,A -85,B 0,C 180,E1 3183.494,E2 3183.494} C_VEL
LIN {X 0,Y 710.247,Z 910.137,A -85,B 0,C 180,E1 3186.598,E2 3186.598} C_VEL
LIN {X 0,Y 712.114,Z 835.785,A -85,B 0,C 180,E1 3188.441,E2 3188.441} C_VEL
LIN {X 0,Y 710.824,Z 786.153,A -85,B 0,C 180,E1 3189.202,E2 3189.202} C_VEL
LIN {X 0,Y 697.959,Z 762.06,A -85,B 0,C 180,E1 3190.583,E2 3190.583} C_VEL
LIN {X 0,Y 698.531,Z 762.06,A -85,B 0,C 180,E1 3196.777,E2 3196.777} C_VEL
LIN {X 0,Y 698.594,Z 762.06,A -85,B 0,C 180,E1 3204.818,E2 3204.818} C_VEL
LIN {X 0,Y 698.733,Z 762.06,A -85,B 0,C 180,E1 3212.128,E2 3212.128} C_VEL
LIN {X 0,Y 698.128,Z 762.06,A -85,B 0,C 180,E1 3218.947,E2 3218.947} C_VEL
LIN {X 0,Y 698.617,Z 762.06,A -85,B 0,C 180,E1 3225.499,E2 3225.499} C_VEL
LIN {X 0,Y 698.727,Z 762.06,A -85,B 0,C 180,E1 3233.104,E2 3233.104} C_VEL
LIN {X 0,Y 698.834,Z 762.06,A -85,B 0,C 180,E1 3240.586,E2 3240.586} C_VEL
LIN {X 0,Y 698.591,Z 762.06,A -85,B 0,C 180,E1 3248.571,E2 3248.571} C_VEL
LIN {X 0,Y 698.721,Z 762.06,A -85,B 0,C 180,E1 3255.712,E2 3255.712} C_VEL
LIN {X 0,Y 698.732,Z 762.06,A -85,B 0,C 180,E1 3263.646,E2 3263.646} C_VEL
LIN {X 0,Y 698.657,Z 762.06,A -85,B 0,C 180,E1 3270.859,E2 3270.859} C_VEL
LIN {X 0,Y 698.365,Z 762.06,A -85,B 0,C 180,E1 3279.477,E2 3279.477} C_VEL
LIN {X 0,Y 698.473,Z 762.06,A -85,B 0,C 180,E1 3286.775,E2 3286.775} C_VEL
LIN {X 0,Y 698.217,Z 763.912,A -85,B 0,C 180,E1 3290.006,E2 3290.006} C_VEL
LIN {X 0,Y 712.281,Z 791.091,A -85,B 0,C 180,E1 3291.298,E2 3291.298} C_VEL
LIN {X 0,Y 710.589,Z 867.693,A -85,B 0,C 180,E1 3292.951,E2 3292.951} C_VEL
LIN {X 0,Y 707.761,Z 940.877,A -85,B 0,C 180,E1 3295.847,E2 3295.847} C_VEL
LIN {X 0,Y 704.495,Z 1010.738,A -85,B 0,C 180,E1 3300.056,E2 3300.056} C_VEL
LIN {X 0,Y 701.737,Z 1070.62,A -85,B 0,C 180,E1 3305.223,E2 3305.223} C_VEL
LIN {X 0,Y 700.038,Z 1116.941,A -85,B 0,C 180,E1 3310.837,E2 3310.837} C_VEL
LIN {X 0,Y 699.219,Z 1149.331,A -85,B 0,C 180,E1 3316.476,E2 3316.476} C_VEL
LIN {X 0,Y 699.25,Z 1169.048,A -85,B 0,C 180,E1 3321.858,E2 3321.858} C_VEL
LIN {X 0,Y 699.453,Z 1178.391,A -85,B 0,C 180,E1 3326.858,E2 3326.858} C_VEL
LIN {X 0,Y 699.404,Z 1178.368,A -85,B 0,C 180,E1 3333.076,E2 3333.076} C_VEL
LIN {X 0,Y 699.223,Z 1165.184,A -85,B 0,C 180,E1 3339.365,E2 3339.365} C_VEL
LIN {X 0,Y 699.645,Z 1139.76,A -85,B 0,C 180,E1 3345.336,E2 3345.336} C_VEL
LIN {X 0,Y 700.766,Z 1099.565,A -85,B 0,C 180,E1 3351.409,E2 3351.409} C_VEL
LIN {X 0,Y 702.974,Z 1046.623,A -85,B 0,C 180,E1 3356.965,E2 3356.965} C_VEL
LIN {X 0,Y 705.944,Z 982.593,A -85,B 0,C 180,E1 3361.737,E2 3361.737} C_VEL
LIN {X 0,Y 709.034,Z 911.809,A -85,B 0,C 180,E1 3365.372,E2 3365.372} C_VEL
LIN {X 0,Y 711.513,Z 837.229,A -85,B 0,C 180,E1 3367.766,E2 3367.766} C_VEL
LIN {X 0,Y 710.639,Z 785.116,A -85,B 0,C 180,E1 3368.8,E2 3368.8} C_VEL
LIN {X 0,Y 698.926,Z 762.06,A -85,B 0,C 180,E1 3370.004,E2 3370.004} C_VEL
LIN {X 0,Y 698.565,Z 762.06,A -85,B 0,C 180,E1 3378.562,E2 3378.562} C_VEL
LIN {X 0,Y 699.428,Z 762.786,A -85,B 0,C 180,E1 3386.24,E2 3386.24} C_VEL
LIN {X 0,Y 700.393,Z 838.391,A -85,B 0,C 180,E1 3389.203,E2 3389.203} C_VEL
LIN {X 0,Y 700.804,Z 969.458,A -85,B 0,C 180,E1 3390.752,E2 3390.752} C_VEL
LIN {X 0,Y 700.249,Z 1008.219,A -85,B 0,C 180,E1 3392.414,E2 3392.414} C_VEL
LIN {X 0,Y 699.642,Z 1038.096,A -85,B 0,C 180,E1 3395.024,E2 3395.024} C_VEL
LIN {X 0,Y 699.398,Z 1055.354,A -85,B 0,C 180,E1 3398.131,E2 3398.131} C_VEL
LIN {X 0,Y 699.497,Z 1059.63,A -85,B 0,C 180,E1 3401.707,E2 3401.707} C_VEL
LIN {X 0,Y 699.791,Z 1049.433,A -85,B 0,C 180,E1 3405.156,E2 3405.156} C_VEL
LIN {X 0,Y 699.914,Z 1026.029,A -85,B 0,C 180,E1 3408.153,E2 3408.153} C_VEL
LIN {X 0,Y 700.546,Z 991.592,A -85,B 0,C 180,E1 3410.377,E2 3410.377} C_VEL
LIN {X 0,Y 700.936,Z 949.103,A -85,B 0,C 180,E1 3411.557,E2 3411.557} C_VEL
LIN {X 0,Y 700.499,Z 832.301,A -85,B 0,C 180,E1 3412.921,E2 3412.921} C_VEL
LIN {X 0,Y 699.785,Z 762.06,A -85,B 0,C 180,E1 3415.684,E2 3415.684} C_VEL
LIN {X 0,Y 699.104,Z 762.06,A -85,B 0,C 180,E1 3425.641,E2 3425.641} C_VEL
LIN {X 0,Y 699.012,Z 762.06,A -85,B 0,C 180,E1 3433.211,E2 3433.211} C_VEL
LIN {X 0,Y 698.483,Z 762.06,A -85,B 0,C 180,E1 3438.199,E2 3438.199} C_VEL
LIN {X 0,Y 690.793,Z 762.06,A -85,B 0,C 180,E1 3441.069,E2 3441.069} C_VEL
LIN {X 0,Y 690.556,Z 762.06,A -85,B 0,C 180,E1 3449.849,E2 3449.849} C_VEL
LIN {X 0,Y 690.587,Z 762.06,A -85,B 0,C 180,E1 3457.217,E2 3457.217} C_VEL
LIN {X 0,Y 690.512,Z 762.06,A -85,B 0,C 180,E1 3466.243,E2 3466.243} C_VEL
LIN {X 0,Y 690.128,Z 763.776,A -85,B 0,C 180,E1 3469.081,E2 3469.081} C_VEL
LIN {X 0,Y 706.003,Z 795.18,A -85,B 0,C 180,E1 3470.594,E2 3470.594} C_VEL
LIN {X 0,Y 704.958,Z 875.584,A -85,B 0,C 180,E1 3471.991,E2 3471.991} C_VEL
LIN {X 0,Y 702.157,Z 946.349,A -85,B 0,C 180,E1 3474.385,E2 3474.385} C_VEL
LIN {X 0,Y 698.535,Z 1017.053,A -85,B 0,C 180,E1 3478.139,E2 3478.139} C_VEL
LIN {X 0,Y 695.164,Z 1079.741,A -85,B 0,C 180,E1 3482.947,E2 3482.947} C_VEL
LIN {X 0,Y 692.706,Z 1131.203,A -85,B 0,C 180,E1 3488.487,E2 3488.487} C_VEL
LIN {X 0,Y 691.564,Z 1166.294,A -85,B 0,C 180,E1 3493.79,E2 3493.79} C_VEL
LIN {X 0,Y 690.983,Z 1192.294,A -85,B 0,C 180,E1 3499.596,E2 3499.596} C_VEL
LIN {X 0,Y 691.008,Z 1205.924,A -85,B 0,C 180,E1 3504.995,E2 3504.995} C_VEL
LIN {X 0,Y 690.901,Z 1209.751,A -85,B 0,C 180,E1 3511.01,E2 3511.01} C_VEL
LIN {X 0,Y 691.008,Z 1203.452,A -85,B 0,C 180,E1 3516.337,E2 3516.337} C_VEL
LIN {X 0,Y 691.237,Z 1185.508,A -85,B 0,C 180,E1 3522.202,E2 3522.202} C_VEL
LIN {X 0,Y 691.925,Z 1154.195,A -85,B 0,C 180,E1 3528.257,E2 3528.257} C_VEL
LIN {X 0,Y 693.846,Z 1109.124,A -85,B 0,C 180,E1 3534.122,E2 3534.122} C_VEL
LIN {X 0,Y 696.787,Z 1050.689,A -85,B 0,C 180,E1 3539.489,E2 3539.489} C_VEL
LIN {X 0,Y 700.407,Z 982.698,A -85,B 0,C 180,E1 3543.874,E2 3543.874} C_VEL
LIN {X 0,Y 703.668,Z 911.895,A -85,B 0,C 180,E1 3546.936,E2 3546.936} C_VEL
LIN {X 0,Y 705.775,Z 837.9,A -85,B 0,C 180,E1 3548.812,E2 3548.812} C_VEL
LIN {X 0,Y 704.737,Z 789.443,A -85,B 0,C 180,E1 3549.564,E2 3549.564} C_VEL
LIN {X 0,Y 690.015,Z 762.06,A -85,B 0,C 180,E1 3551.054,E2 3551.054} C_VEL
LIN {X 0,Y 690.251,Z 762.06,A -85,B 0,C 180,E1 3557.85,E2 3557.85} C_VEL
LIN {X 0,Y 690.517,Z 762.06,A -85,B 0,C 180,E1 3565.879,E2 3565.879} C_VEL
LIN {X 0,Y 690.749,Z 762.06,A -85,B 0,C 180,E1 3573.196,E2 3573.196} C_VEL
LIN {X 0,Y 690.294,Z 762.06,A -85,B 0,C 180,E1 3581.376,E2 3581.376} C_VEL
LIN {X 0,Y 690.22,Z 762.06,A -85,B 0,C 180,E1 3588.193,E2 3588.193} C_VEL
LIN {X 0,Y 690.367,Z 762.06,A -85,B 0,C 180,E1 3594.287,E2 3594.287} C_VEL
LIN {X 0,Y 690.827,Z 762.06,A -85,B 0,C 180,E1 3600.592,E2 3600.592} C_VEL
LIN {X 0,Y 690.761,Z 762.06,A -85,B 0,C 180,E1 3608.171,E2 3608.171} C_VEL
LIN {X 0,Y 690.619,Z 762.06,A -85,B 0,C 180,E1 3615.901,E2 3615.901} C_VEL
LIN {X 0,Y 690.564,Z 762.06,A -85,B 0,C 180,E1 3624.156,E2 3624.156} C_VEL
LIN {X 0,Y 690.386,Z 762.06,A -85,B 0,C 180,E1 3632.141,E2 3632.141} C_VEL
LIN {X 0,Y 690.511,Z 762.06,A -85,B 0,C 180,E1 3638.725,E2 3638.725} C_VEL
LIN {X 0,Y 690.557,Z 762.06,A -85,B 0,C 180,E1 3646.154,E2 3646.154} C_VEL
LIN {X 0,Y 690.165,Z 763.844,A -85,B 0,C 180,E1 3649.443,E2 3649.443} C_VEL
LIN {X 0,Y 706.004,Z 795.159,A -85,B 0,C 180,E1 3650.952,E2 3650.952} C_VEL
LIN {X 0,Y 703.99,Z 871.024,A -85,B 0,C 180,E1 3652.662,E2 3652.662} C_VEL
LIN {X 0,Y 700.832,Z 944.067,A -85,B 0,C 180,E1 3655.627,E2 3655.627} C_VEL
LIN {X 0,Y 697.094,Z 1013.527,A -85,B 0,C 180,E1 3659.92,E2 3659.92} C_VEL
LIN {X 0,Y 694.027,Z 1072.665,A -85,B 0,C 180,E1 3665.147,E2 3665.147} C_VEL
LIN {X 0,Y 692.13,Z 1118.405,A -85,B 0,C 180,E1 3670.83,E2 3670.83} C_VEL
LIN {X 0,Y 691.162,Z 1150.807,A -85,B 0,C 180,E1 3676.639,E2 3676.639} C_VEL
LIN {X 0,Y 691.05,Z 1170.675,A -85,B 0,C 180,E1 3682.396,E2 3682.396} C_VEL
LIN {X 0,Y 690.895,Z 1179.399,A -85,B 0,C 180,E1 3688.079,E2 3688.079} C_VEL
LIN {X 0,Y 691.19,Z 1177.93,A -85,B 0,C 180,E1 3693.496,E2 3693.496} C_VEL
LIN {X 0,Y 691.205,Z 1165.289,A -85,B 0,C 180,E1 3699.442,E2 3699.442} C_VEL
LIN {X 0,Y 691.598,Z 1139.056,A -85,B 0,C 180,E1 3705.65,E2 3705.65} C_VEL
LIN {X 0,Y 692.988,Z 1099.059,A -85,B 0,C 180,E1 3711.726,E2 3711.726} C_VEL
LIN {X 0,Y 695.546,Z 1045.24,A -85,B 0,C 180,E1 3717.404,E2 3717.404} C_VEL
LIN {X 0,Y 698.959,Z 980.591,A -85,B 0,C 180,E1 3722.226,E2 3722.226} C_VEL
LIN {X 0,Y 702.473,Z 909.912,A -85,B 0,C 180,E1 3725.839,E2 3725.839} C_VEL
LIN {X 0,Y 705.13,Z 837.066,A -85,B 0,C 180,E1 3728.173,E2 3728.173} C_VEL
LIN {X 0,Y 704.484,Z 788.283,A -85,B 0,C 180,E1 3729.161,E2 3729.161} C_VEL
LIN {X 0,Y 690.976,Z 762.06,A -85,B 0,C 180,E1 3730.538,E2 3730.538} C_VEL
LIN {X 0,Y 690.77,Z 762.06,A -85,B 0,C 180,E1 3739.661,E2 3739.661} C_VEL
LIN {X 0,Y 691.467,Z 763.463,A -85,B 0,C 180,E1 3746.09,E2 3746.09} C_VEL
LIN {X 0,Y 693.048,Z 833.956,A -85,B 0,C 180,E1 3748.908,E2 3748.908} C_VEL
LIN {X 0,Y 692.973,Z 970.622,A -85,B 0,C 180,E1 3750.657,E2 3750.657} C_VEL
LIN {X 0,Y 692.363,Z 1008.995,A -85,B 0,C 180,E1 3752.337,E2 3752.337} C_VEL
LIN {X 0,Y 691.685,Z 1037.992,A -85,B 0,C 180,E1 3754.914,E2 3754.914} C_VEL
LIN {X 0,Y 691.4,Z 1055.465,A -85,B 0,C 180,E1 3758.131,E2 3758.131} C_VEL
LIN {X 0,Y 691.468,Z 1059.75,A -85,B 0,C 180,E1 3761.487,E2 3761.487} C_VEL
LIN {X 0,Y 691.741,Z 1050.344,A -85,B 0,C 180,E1 3765.019,E2 3765.019} C_VEL
LIN {X 0,Y 691.995,Z 1027.051,A -85,B 0,C 180,E1 3768.176,E2 3768.176} C_VEL
LIN {X 0,Y 692.673,Z 992.669,A -85,B 0,C 180,E1 3770.463,E2 3770.463} C_VEL
LIN {X 0,Y 693.103,Z 950.366,A -85,B 0,C 180,E1 3771.659,E2 3771.659} C_VEL
LIN {X 0,Y 692.715,Z 833.584,A -85,B 0,C 180,E1 3773.039,E2 3773.039} C_VEL
LIN {X 0,Y 691.784,Z 762.06,A -85,B 0,C 180,E1 3775.867,E2 3775.867} C_VEL
LIN {X 0,Y 691.083,Z 762.06,A -85,B 0,C 180,E1 3785.707,E2 3785.707} C_VEL
LIN {X 0,Y 690.928,Z 762.06,A -85,B 0,C 180,E1 3793.369,E2 3793.369} C_VEL
LIN {X 0,Y 690.793,Z 762.06,A -85,B 0,C 180,E1 3801.069,E2 3801.069} C_VEL
LIN {X 0,Y 681.985,Z 762.06,A -85,B 0,C 180,E1 3803.946,E2 3803.946} C_VEL
LIN {X 0,Y 682.216,Z 762.06,A -85,B 0,C 180,E1 3811.163,E2 3811.163} C_VEL
LIN {X 0,Y 682.324,Z 762.06,A -85,B 0,C 180,E1 3817.922,E2 3817.922} C_VEL
LIN {X 0,Y 682.482,Z 762.06,A -85,B 0,C 180,E1 3826.317,E2 3826.317} C_VEL
LIN {X 0,Y 682.191,Z 763.83,A -85,B 0,C 180,E1 3828.501,E2 3828.501} C_VEL
LIN {X 0,Y 699.803,Z 798.419,A -85,B 0,C 180,E1 3830.218,E2 3830.218} C_VEL
LIN {X 0,Y 698.539,Z 877.24,A -85,B 0,C 180,E1 3831.624,E2 3831.624} C_VEL
LIN {X 0,Y 695.39,Z 948.346,A -85,B 0,C 180,E1 3834.076,E2 3834.076} C_VEL
LIN {X 0,Y 691.375,Z 1018.774,A -85,B 0,C 180,E1 3837.885,E2 3837.885} C_VEL
LIN {X 0,Y 687.57,Z 1081.957,A -85,B 0,C 180,E1 3842.832,E2 3842.832} C_VEL
LIN {X 0,Y 684.863,Z 1132.902,A -85,B 0,C 180,E1 3848.451,E2 3848.451} C_VEL
LIN {X 0,Y 683.561,Z 1168.062,A -85,B 0,C 180,E1 3853.926,E2 3853.926} C_VEL
LIN {X 0,Y 683.028,Z 1192.295,A -85,B 0,C 180,E1 3859.474,E2 3859.474} C_VEL
LIN {X 0,Y 683.035,Z 1205.923,A -85,B 0,C 180,E1 3864.936,E2 3864.936} C_VEL
LIN {X 0,Y 683.01,Z 1209.847,A -85,B 0,C 180,E1 3870.67,E2 3870.67} C_VEL
LIN {X 0,Y 682.983,Z 1203.452,A -85,B 0,C 180,E1 3876.412,E2 3876.412} C_VEL
LIN {X 0,Y 683.269,Z 1186.055,A -85,B 0,C 180,E1 3882.214,E2 3882.214} C_VEL
LIN {X 0,Y 684.046,Z 1155.306,A -85,B 0,C 180,E1 3888.295,E2 3888.295} C_VEL
LIN {X 0,Y 686.096,Z 1111.045,A -85,B 0,C 180,E1 3894.187,E2 3894.187} C_VEL
LIN {X 0,Y 689.375,Z 1053.301,A -85,B 0,C 180,E1 3899.625,E2 3899.625} C_VEL
LIN {X 0,Y 693.37,Z 985.99,A -85,B 0,C 180,E1 3904.081,E2 3904.081} C_VEL
LIN {X 0,Y 697.136,Z 912.939,A -85,B 0,C 180,E1 3907.304,E2 3907.304} C_VEL
LIN {X 0,Y 699.519,Z 838.367,A -85,B 0,C 180,E1 3909.216,E2 3909.216} C_VEL
LIN {X 0,Y 698.342,Z 792.523,A -85,B 0,C 180,E1 3909.959,E2 3909.959} C_VEL
LIN {X 0,Y 682.082,Z 762.06,A -85,B 0,C 180,E1 3911.585,E2 3911.585} C_VEL
LIN {X 0,Y 682.202,Z 762.06,A -85,B 0,C 180,E1 3918.948,E2 3918.948} C_VEL
LIN {X 0,Y 682.596,Z 762.06,A -85,B 0,C 180,E1 3926.96,E2 3926.96} C_VEL
LIN {X 0,Y 682.967,Z 762.06,A -85,B 0,C 180,E1 3935.692,E2 3935.692} C_VEL
LIN {X 0,Y 682.668,Z 762.06,A -85,B 0,C 180,E1 3945.34,E2 3945.34} C_VEL
LIN {X 0,Y 682.778,Z 762.06,A -85,B 0,C 180,E1 3952.942,E2 3952.942} C_VEL
LIN {X 0,Y 682.82,Z 762.06,A -85,B 0,C 180,E1 3960.599,E2 3960.599} C_VEL
LIN {X 0,Y 682.712,Z 762.06,A -85,B 0,C 180,E1 3968.268,E2 3968.268} C_VEL
LIN {X 0,Y 682.536,Z 762.06,A -85,B 0,C 180,E1 3976.094,E2 3976.094} C_VEL
LIN {X 0,Y 682.551,Z 762.06,A -85,B 0,C 180,E1 3984.242,E2 3984.242} C_VEL
LIN {X 0,Y 682.516,Z 762.06,A -85,B 0,C 180,E1 3991.45,E2 3991.45} C_VEL
LIN {X 0,Y 682.333,Z 762.06,A -85,B 0,C 180,E1 3999.278,E2 3999.278} C_VEL
LIN {X 0,Y 682.275,Z 762.06,A -85,B 0,C 180,E1 4007.243,E2 4007.243} C_VEL
LIN {X 0,Y 682.162,Z 763.884,A -85,B 0,C 180,E1 4008.866,E2 4008.866} C_VEL
LIN {X 0,Y 699.746,Z 797.773,A -85,B 0,C 180,E1 4010.577,E2 4010.577} C_VEL
LIN {X 0,Y 697.449,Z 872.654,A -85,B 0,C 180,E1 4012.309,E2 4012.309} C_VEL
LIN {X 0,Y 693.876,Z 946.122,A -85,B 0,C 180,E1 4015.35,E2 4015.35} C_VEL
LIN {X 0,Y 689.752,Z 1014.998,A -85,B 0,C 180,E1 4019.683,E2 4019.683} C_VEL
LIN {X 0,Y 686.383,Z 1073.792,A -85,B 0,C 180,E1 4024.973,E2 4024.973} C_VEL
LIN {X 0,Y 684.267,Z 1119.326,A -85,B 0,C 180,E1 4030.742,E2 4030.742} C_VEL
LIN {X 0,Y 683.255,Z 1150.806,A -85,B 0,C 180,E1 4036.481,E2 4036.481} C_VEL
LIN {X 0,Y 683.09,Z 1170.671,A -85,B 0,C 180,E1 4042.307,E2 4042.307} C_VEL
LIN {X 0,Y 682.909,Z 1179.396,A -85,B 0,C 180,E1 4048.056,E2 4048.056} C_VEL
LIN {X 0,Y 683.366,Z 1178.37,A -85,B 0,C 180,E1 4053.148,E2 4053.148} C_VEL
LIN {X 0,Y 683.173,Z 1165.291,A -85,B 0,C 180,E1 4059.555,E2 4059.555} C_VEL
LIN {X 0,Y 683.662,Z 1140.124,A -85,B 0,C 180,E1 4065.636,E2 4065.636} C_VEL
LIN {X 0,Y 685.176,Z 1100.209,A -85,B 0,C 180,E1 4071.841,E2 4071.841} C_VEL
LIN {X 0,Y 687.985,Z 1047.3,A -85,B 0,C 180,E1 4077.541,E2 4077.541} C_VEL
LIN {X 0,Y 691.808,Z 982.624,A -85,B 0,C 180,E1 4082.464,E2 4082.464} C_VEL
LIN {X 0,Y 695.748,Z 911.708,A -85,B 0,C 180,E1 4086.159,E2 4086.159} C_VEL
LIN {X 0,Y 698.751,Z 838.976,A -85,B 0,C 180,E1 4088.537,E2 4088.537} C_VEL
LIN {X 0,Y 698.313,Z 791.775,A -85,B 0,C 180,E1 4089.523,E2 4089.523} C_VEL
LIN {X 0,Y 682.938,Z 762.06,A -85,B 0,C 180,E1 4091.103,E2 4091.103} C_VEL
LIN {X 0,Y 682.803,Z 762.06,A -85,B 0,C 180,E1 4100.754,E2 4100.754} C_VEL
LIN {X 0,Y 683.343,Z 762.987,A -85,B 0,C 180,E1 4105.891,E2 4105.891} C_VEL
LIN {X 0,Y 685.372,Z 813.312,A -85,B 0,C 180,E1 4107.942,E2 4107.942} C_VEL
LIN {X 0,Y 684.703,Z 847.694,A -85,B 0,C 180,E1 4109.036,E2 4109.036} C_VEL
LIN {X 0,Y 685.142,Z 970.909,A -85,B 0,C 180,E1 4110.532,E2 4110.532} C_VEL
LIN {X 0,Y 684.517,Z 1009.641,A -85,B 0,C 180,E1 4112.224,E2 4112.224} C_VEL
LIN {X 0,Y 683.806,Z 1039.838,A -85,B 0,C 180,E1 4114.961,E2 4114.961} C_VEL
LIN {X 0,Y 683.511,Z 1056.792,A -85,B 0,C 180,E1 4118.213,E2 4118.213} C_VEL
LIN {X 0,Y 683.52,Z 1060.792,A -85,B 0,C 180,E1 4121.264,E2 4121.264} C_VEL
LIN {X 0,Y 683.824,Z 1051.726,A -85,B 0,C 180,E1 4125.007,E2 4125.007} C_VEL
LIN {X 0,Y 684.156,Z 1028.698,A -85,B 0,C 180,E1 4128.201,E2 4128.201} C_VEL
LIN {X 0,Y 684.821,Z 993.931,A -85,B 0,C 180,E1 4130.553,E2 4130.553} C_VEL
LIN {X 0,Y 685.233,Z 951.682,A -85,B 0,C 180,E1 4131.763,E2 4131.763} C_VEL
LIN {X 0,Y 684.934,Z 834.875,A -85,B 0,C 180,E1 4133.159,E2 4133.159} C_VEL
LIN {X 0,Y 683.789,Z 762.06,A -85,B 0,C 180,E1 4136.12,E2 4136.12} C_VEL
LIN {X 0,Y 683.034,Z 762.06,A -85,B 0,C 180,E1 4145.774,E2 4145.774} C_VEL
LIN {X 0,Y 682.836,Z 762.06,A -85,B 0,C 180,E1 4153.53,E2 4153.53} C_VEL
LIN {X 0,Y 682.581,Z 762.06,A -85,B 0,C 180,E1 4161.556,E2 4161.556} C_VEL
LIN {X 0,Y 681.985,Z 762.06,A -85,B 0,C 180,E1 4163.946,E2 4163.946} C_VEL
LIN {X 0,Y 674.401,Z 762.06,A -85,B 0,C 180,E1 4166.868,E2 4166.868} C_VEL
LIN {X 0,Y 674.378,Z 762.06,A -85,B 0,C 180,E1 4175.056,E2 4175.056} C_VEL
LIN {X 0,Y 674.595,Z 762.06,A -85,B 0,C 180,E1 4184.934,E2 4184.934} C_VEL
LIN {X 0,Y 674.195,Z 763.189,A -85,B 0,C 180,E1 4187.888,E2 4187.888} C_VEL
LIN {X 0,Y 693.638,Z 800.59,A -85,B 0,C 180,E1 4189.822,E2 4189.822} C_VEL
LIN {X 0,Y 692.166,Z 878.433,A -85,B 0,C 180,E1 4191.239,E2 4191.239} C_VEL
LIN {X 0,Y 688.751,Z 948.19,A -85,B 0,C 180,E1 4193.668,E2 4193.668} C_VEL
LIN {X 0,Y 684.3,Z 1018.776,A -85,B 0,C 180,E1 4197.512,E2 4197.512} C_VEL
LIN {X 0,Y 680.075,Z 1082.427,A -85,B 0,C 180,E1 4202.553,E2 4202.553} C_VEL
LIN {X 0,Y 677.21,Z 1132.695,A -85,B 0,C 180,E1 4208.167,E2 4208.167} C_VEL
LIN {X 0,Y 675.695,Z 1168.064,A -85,B 0,C 180,E1 4213.734,E2 4213.734} C_VEL
LIN {X 0,Y 675.008,Z 1193.376,A -85,B 0,C 180,E1 4219.675,E2 4219.675} C_VEL
LIN {X 0,Y 674.832,Z 1206.868,A -85,B 0,C 180,E1 4225.521,E2 4225.521} C_VEL
LIN {X 0,Y 675.031,Z 1209.849,A -85,B 0,C 180,E1 4230.678,E2 4230.678} C_VEL
LIN {X 0,Y 674.987,Z 1203.453,A -85,B 0,C 180,E1 4236.488,E2 4236.488} C_VEL
LIN {X 0,Y 675.271,Z 1186.055,A -85,B 0,C 180,E1 4242.36,E2 4242.36} C_VEL
LIN {X 0,Y 676.128,Z 1156.3,A -85,B 0,C 180,E1 4248.347,E2 4248.347} C_VEL
LIN {X 0,Y 678.373,Z 1112.984,A -85,B 0,C 180,E1 4254.25,E2 4254.25} C_VEL
LIN {X 0,Y 681.915,Z 1056.406,A -85,B 0,C 180,E1 4259.725,E2 4259.725} C_VEL
LIN {X 0,Y 686.278,Z 989.546,A -85,B 0,C 180,E1 4264.271,E2 4264.271} C_VEL
LIN {X 0,Y 690.372,Z 918.453,A -85,B 0,C 180,E1 4267.518,E2 4267.518} C_VEL
LIN {X 0,Y 693.175,Z 842.529,A -85,B 0,C 180,E1 4269.563,E2 4269.563} C_VEL
LIN {X 0,Y 692.293,Z 796.005,A -85,B 0,C 180,E1 4270.333,E2 4270.333} C_VEL
LIN {X 0,Y 674.177,Z 762.06,A -85,B 0,C 180,E1 4272.177,E2 4272.177} C_VEL
LIN {X 0,Y 674.314,Z 762.06,A -85,B 0,C 180,E1 4280.064,E2 4280.064} C_VEL
LIN {X 0,Y 674.72,Z 762.06,A -85,B 0,C 180,E1 4288.055,E2 4288.055} C_VEL
LIN {X 0,Y 674.983,Z 762.06,A -85,B 0,C 180,E1 4295.647,E2 4295.647} C_VEL
LIN {X 0,Y 674.711,Z 762.06,A -85,B 0,C 180,E1 4304.974,E2 4304.974} C_VEL
LIN {X 0,Y 674.796,Z 762.06,A -85,B 0,C 180,E1 4312.858,E2 4312.858} C_VEL
LIN {X 0,Y 674.832,Z 762.06,A -85,B 0,C 180,E1 4320.606,E2 4320.606} C_VEL
LIN {X 0,Y 674.667,Z 762.06,A -85,B 0,C 180,E1 4328.367,E2 4328.367} C_VEL
LIN {X 0,Y 674.448,Z 762.06,A -85,B 0,C 180,E1 4336.293,E2 4336.293} C_VEL
LIN {X 0,Y 674.488,Z 762.06,A -85,B 0,C 180,E1 4344.55,E2 4344.55} C_VEL
LIN {X 0,Y 674.299,Z 762.06,A -85,B 0,C 180,E1 4352.388,E2 4352.388} C_VEL
LIN {X 0,Y 674.267,Z 762.06,A -85,B 0,C 180,E1 4359.841,E2 4359.841} C_VEL
LIN {X 0,Y 674.336,Z 762.06,A -85,B 0,C 180,E1 4366.936,E2 4366.936} C_VEL
LIN {X 0,Y 674.25,Z 763.828,A -85,B 0,C 180,E1 4368.277,E2 4368.277} C_VEL
LIN {X 0,Y 693.54,Z 800.645,A -85,B 0,C 180,E1 4370.2,E2 4370.2} C_VEL
LIN {X 0,Y 690.93,Z 874.557,A -85,B 0,C 180,E1 4371.959,E2 4371.959} C_VEL
LIN {X 0,Y 687.006,Z 947.082,A -85,B 0,C 180,E1 4375.008,E2 4375.008} C_VEL
LIN {X 0,Y 682.514,Z 1015.69,A -85,B 0,C 180,E1 4379.383,E2 4379.383} C_VEL
LIN {X 0,Y 678.764,Z 1074.73,A -85,B 0,C 180,E1 4384.776,E2 4384.776} C_VEL
LIN {X 0,Y 676.454,Z 1119.682,A -85,B 0,C 180,E1 4390.566,E2 4390.566} C_VEL
LIN {X 0,Y 675.37,Z 1150.804,A -85,B 0,C 180,E1 4396.32,E2 4396.32} C_VEL
LIN {X 0,Y 675.137,Z 1170.667,A -85,B 0,C 180,E1 4402.216,E2 4402.216} C_VEL
LIN {X 0,Y 674.921,Z 1179.392,A -85,B 0,C 180,E1 4408.033,E2 4408.033} C_VEL
LIN {X 0,Y 675.343,Z 1178.371,A -85,B 0,C 180,E1 4413.186,E2 4413.186} C_VEL
LIN {X 0,Y 675.129,Z 1165.294,A -85,B 0,C 180,E1 4419.669,E2 4419.669} C_VEL
LIN {X 0,Y 675.69,Z 1139.865,A -85,B 0,C 180,E1 4425.876,E2 4425.876} C_VEL
LIN {X 0,Y 677.391,Z 1101.042,A -85,B 0,C 180,E1 4431.999,E2 4431.999} C_VEL
LIN {X 0,Y 680.47,Z 1048.279,A -85,B 0,C 180,E1 4437.781,E2 4437.781} C_VEL
LIN {X 0,Y 684.702,Z 984.036,A -85,B 0,C 180,E1 4442.748,E2 4442.748} C_VEL
LIN {X 0,Y 689.025,Z 913.542,A -85,B 0,C 180,E1 4446.485,E2 4446.485} C_VEL
LIN {X 0,Y 692.413,Z 840.151,A -85,B 0,C 180,E1 4448.925,E2 4448.925} C_VEL
LIN {X 0,Y 692.166,Z 795.094,A -85,B 0,C 180,E1 4449.892,E2 4449.892} C_VEL
LIN {X 0,Y 674.904,Z 762.06,A -85,B 0,C 180,E1 4451.716,E2 4451.716} C_VEL
LIN {X 0,Y 674.792,Z 762.06,A -85,B 0,C 180,E1 4460.82,E2 4460.82} C_VEL
LIN {X 0,Y 675.468,Z 763.954,A -85,B 0,C 180,E1 4465.751,E2 4465.751} C_VEL
LIN {X 0,Y 677.592,Z 810.405,A -85,B 0,C 180,E1 4467.653,E2 4467.653} C_VEL
LIN {X 0,Y 676.879,Z 847.322,A -85,B 0,C 180,E1 4468.896,E2 4468.896} C_VEL
LIN {X 0,Y 677.306,Z 971.215,A -85,B 0,C 180,E1 4470.406,E2 4470.406} C_VEL
LIN {X 0,Y 676.652,Z 1010.055,A -85,B 0,C 180,E1 4472.099,E2 4472.099} C_VEL
LIN {X 0,Y 675.905,Z 1040.798,A -85,B 0,C 180,E1 4474.892,E2 4474.892} C_VEL
LIN {X 0,Y 675.601,Z 1058.144,A -85,B 0,C 180,E1 4478.291,E2 4478.291} C_VEL
LIN {X 0,Y 675.596,Z 1062.008,A -85,B 0,C 180,E1 4481.036,E2 4481.036} C_VEL
LIN {X 0,Y 675.828,Z 1053.927,A -85,B 0,C 180,E1 4484.825,E2 4484.825} C_VEL
LIN {X 0,Y 676.334,Z 1032.01,A -85,B 0,C 180,E1 4488.062,E2 4488.062} C_VEL
LIN {X 0,Y 676.972,Z 999.267,A -85,B 0,C 180,E1 4490.443,E2 4490.443} C_VEL
LIN {X 0,Y 677.361,Z 958.046,A -85,B 0,C 180,E1 4491.788,E2 4491.788} C_VEL
LIN {X 0,Y 677.191,Z 836.138,A -85,B 0,C 180,E1 4493.283,E2 4493.283} C_VEL
LIN {X 0,Y 675.801,Z 762.06,A -85,B 0,C 180,E1 4496.288,E2 4496.288} C_VEL
LIN {X 0,Y 674.997,Z 762.06,A -85,B 0,C 180,E1 4505.843,E2 4505.843} C_VEL
LIN {X 0,Y 674.75,Z 762.06,A -85,B 0,C 180,E1 4513.696,E2 4513.696} C_VEL
LIN {X 0,Y 674.477,Z 762.06,A -85,B 0,C 180,E1 4521.829,E2 4521.829} C_VEL
LIN {X 0,Y 674.401,Z 762.06,A -85,B 0,C 180,E1 4526.868,E2 4526.868} C_VEL
LIN {X 0,Y 666.434,Z 762.06,A -85,B 0,C 180,E1 4529.837,E2 4529.837} C_VEL
LIN {X 0,Y 666.231,Z 762.06,A -85,B 0,C 180,E1 4538.267,E2 4538.267} C_VEL
LIN {X 0,Y 666.291,Z 762.06,A -85,B 0,C 180,E1 4547.249,E2 4547.249} C_VEL
LIN {X 0,Y 687.53,Z 803.032,A -85,B 0,C 180,E1 4549.424,E2 4549.424} C_VEL
LIN {X 0,Y 685.757,Z 880.86,A -85,B 0,C 180,E1 4550.878,E2 4550.878} C_VEL
LIN {X 0,Y 681.995,Z 950.934,A -85,B 0,C 180,E1 4553.381,E2 4553.381} C_VEL
LIN {X 0,Y 677.096,Z 1021.575,A -85,B 0,C 180,E1 4557.316,E2 4557.316} C_VEL
LIN {X 0,Y 672.463,Z 1085.151,A -85,B 0,C 180,E1 4562.486,E2 4562.486} C_VEL
LIN {X 0,Y 669.206,Z 1135.636,A -85,B 0,C 180,E1 4568.304,E2 4568.304} C_VEL
LIN {X 0,Y 667.689,Z 1169.832,A -85,B 0,C 180,E1 4573.872,E2 4573.872} C_VEL
LIN {X 0,Y 667.068,Z 1193.375,A -85,B 0,C 180,E1 4579.551,E2 4579.551} C_VEL
LIN {X 0,Y 666.847,Z 1206.867,A -85,B 0,C 180,E1 4585.467,E2 4585.467} C_VEL
LIN {X 0,Y 667.026,Z 1209.851,A -85,B 0,C 180,E1 4590.686,E2 4590.686} C_VEL
LIN {X 0,Y 666.974,Z 1203.453,A -85,B 0,C 180,E1 4596.566,E2 4596.566} C_VEL
LIN {X 0,Y 667.255,Z 1186.054,A -85,B 0,C 180,E1 4602.511,E2 4602.511} C_VEL
LIN {X 0,Y 668.156,Z 1156.303,A -85,B 0,C 180,E1 4608.574,E2 4608.574} C_VEL
LIN {X 0,Y 670.667,Z 1114.008,A -85,B 0,C 180,E1 4614.424,E2 4614.424} C_VEL
LIN {X 0,Y 674.583,Z 1057.238,A -85,B 0,C 180,E1 4620.01,E2 4620.01} C_VEL
LIN {X 0,Y 679.402,Z 990.192,A -85,B 0,C 180,E1 4624.627,E2 4624.627} C_VEL
LIN {X 0,Y 683.929,Z 918.662,A -85,B 0,C 180,E1 4627.925,E2 4627.925} C_VEL
LIN {X 0,Y 686.974,Z 843.025,A -85,B 0,C 180,E1 4629.981,E2 4629.981} C_VEL
LIN {X 0,Y 686.173,Z 799.159,A -85,B 0,C 180,E1 4630.726,E2 4630.726} C_VEL
LIN {X 0,Y 666.318,Z 762.06,A -85,B 0,C 180,E1 4632.81,E2 4632.81} C_VEL
LIN {X 0,Y 666.534,Z 762.06,A -85,B 0,C 180,E1 4641.811,E2 4641.811} C_VEL
LIN {X 0,Y 666.793,Z 762.06,A -85,B 0,C 180,E1 4650.667,E2 4650.667} C_VEL
LIN {X 0,Y 666.321,Z 762.06,A -85,B 0,C 180,E1 4657.89,E2 4657.89} C_VEL
LIN {X 0,Y 666.385,Z 762.06,A -85,B 0,C 180,E1 4666.129,E2 4666.129} C_VEL
LIN {X 0,Y 666.811,Z 762.06,A -85,B 0,C 180,E1 4672.772,E2 4672.772} C_VEL
LIN {X 0,Y 666.825,Z 762.06,A -85,B 0,C 180,E1 4680.614,E2 4680.614} C_VEL
LIN {X 0,Y 666.624,Z 762.06,A -85,B 0,C 180,E1 4688.469,E2 4688.469} C_VEL
LIN {X 0,Y 666.372,Z 762.06,A -85,B 0,C 180,E1 4696.496,E2 4696.496} C_VEL
LIN {X 0,Y 666.418,Z 762.06,A -85,B 0,C 180,E1 4704.868,E2 4704.868} C_VEL
LIN {X 0,Y 666.329,Z 762.06,A -85,B 0,C 180,E1 4712.306,E2 4712.306} C_VEL
LIN {X 0,Y 666.191,Z 762.06,A -85,B 0,C 180,E1 4720.423,E2 4720.423} C_VEL
LIN {X 0,Y 666.375,Z 763.979,A -85,B 0,C 180,E1 4727.673,E2 4727.673} C_VEL
LIN {X 0,Y 687.322,Z 804.852,A -85,B 0,C 180,E1 4729.839,E2 4729.839} C_VEL
LIN {X 0,Y 684.366,Z 878.13,A -85,B 0,C 180,E1 4731.66,E2 4731.66} C_VEL
LIN {X 0,Y 680.032,Z 950.271,A -85,B 0,C 180,E1 4734.781,E2 4734.781} C_VEL
LIN {X 0,Y 675.046,Z 1019.219,A -85,B 0,C 180,E1 4739.296,E2 4739.296} C_VEL
LIN {X 0,Y 671.002,Z 1077.344,A -85,B 0,C 180,E1 4744.753,E2 4744.753} C_VEL
LIN {X 0,Y 668.587,Z 1120.626,A -85,B 0,C 180,E1 4750.476,E2 4750.476} C_VEL
LIN {X 0,Y 667.307,Z 1152.159,A -85,B 0,C 180,E1 4756.487,E2 4756.487} C_VEL
LIN {X 0,Y 667.198,Z 1170.663,A -85,B 0,C 180,E1 4762.123,E2 4762.123} C_VEL
LIN {X 0,Y 666.927,Z 1179.389,A -85,B 0,C 180,E1 4768.01,E2 4768.01} C_VEL
LIN {X 0,Y 667.319,Z 1178.371,A -85,B 0,C 180,E1 4773.224,E2 4773.224} C_VEL
LIN {X 0,Y 667.096,Z 1165.296,A -85,B 0,C 180,E1 4779.787,E2 4779.787} C_VEL
LIN {X 0,Y 667.773,Z 1141.226,A -85,B 0,C 180,E1 4785.807,E2 4785.807} C_VEL
LIN {X 0,Y 669.591,Z 1102.382,A -85,B 0,C 180,E1 4792.094,E2 4792.094} C_VEL
LIN {X 0,Y 672.934,Z 1050.516,A -85,B 0,C 180,E1 4797.908,E2 4797.908} C_VEL
LIN {X 0,Y 677.562,Z 986.087,A -85,B 0,C 180,E1 4802.996,E2 4802.996} C_VEL
LIN {X 0,Y 682.37,Z 914.855,A -85,B 0,C 180,E1 4806.838,E2 4806.838} C_VEL
LIN {X 0,Y 686.12,Z 841.267,A -85,B 0,C 180,E1 4809.321,E2 4809.321} C_VEL
LIN {X 0,Y 686.065,Z 798.228,A -85,B 0,C 180,E1 4810.269,E2 4810.269} C_VEL
LIN {X 0,Y 666.79,Z 762.06,A -85,B 0,C 180,E1 4812.366,E2 4812.366} C_VEL
LIN {X 0,Y 666.732,Z 762.06,A -85,B 0,C 180,E1 4821.678,E2 4821.678} C_VEL
LIN {X 0,Y 667.16,Z 762.633,A -85,B 0,C 180,E1 4825.498,E2 4825.498} C_VEL
LIN {X 0,Y 669.968,Z 801.631,A -85,B 0,C 180,E1 4827.123,E2 4827.123} C_VEL
LIN {X 0,Y 669.08,Z 848.11,A -85,B 0,C 180,E1 4828.765,E2 4828.765} C_VEL
LIN {X 0,Y 669.456,Z 973.88,A -85,B 0,C 180,E1 4830.342,E2 4830.342} C_VEL
LIN {X 0,Y 668.797,Z 1012.808,A -85,B 0,C 180,E1 4832.122,E2 4832.122} C_VEL
LIN {X 0,Y 668.039,Z 1041.078,A -85,B 0,C 180,E1 4834.731,E2 4834.731} C_VEL
LIN {X 0,Y 667.651,Z 1058.539,A -85,B 0,C 180,E1 4838.019,E2 4838.019} C_VEL
LIN {X 0,Y 667.693,Z 1063.077,A -85,B 0,C 180,E1 4840.802,E2 4840.802} C_VEL
LIN {X 0,Y 667.794,Z 1056.204,A -85,B 0,C 180,E1 4844.579,E2 4844.579} C_VEL
LIN {X 0,Y 668.473,Z 1035.066,A -85,B 0,C 180,E1 4847.92,E2 4847.92} C_VEL
LIN {X 0,Y 669.099,Z 1003.844,A -85,B 0,C 180,E1 4850.354,E2 4850.354} C_VEL
LIN {X 0,Y 669.483,Z 963.949,A -85,B 0,C 180,E1 4851.814,E2 4851.814} C_VEL
LIN {X 0,Y 669.424,Z 837.406,A -85,B 0,C 180,E1 4853.409,E2 4853.409} C_VEL
LIN {X 0,Y 667.844,Z 762.079,A -85,B 0,C 180,E1 4856.413,E2 4856.413} C_VEL
LIN {X 0,Y 666.948,Z 762.06,A -85,B 0,C 180,E1 4865.914,E2 4865.914} C_VEL
LIN {X 0,Y 666.668,Z 762.06,A -85,B 0,C 180,E1 4873.865,E2 4873.865} C_VEL
LIN {X 0,Y 666.366,Z 762.06,A -85,B 0,C 180,E1 4882.108,E2 4882.108} C_VEL
LIN {X 0,Y 666.434,Z 762.06,A -85,B 0,C 180,E1 4889.837,E2 4889.837} C_VEL
LIN {X 0,Y 658.066,Z 762.06,A -85,B 0,C 180,E1 4892.818,E2 4892.818} C_VEL
LIN {X 0,Y 657.921,Z 762.06,A -85,B 0,C 180,E1 4899.468,E2 4899.468} C_VEL
LIN {X 0,Y 658.492,Z 763.174,A -85,B 0,C 180,E1 4906.64,E2 4906.64} C_VEL
LIN {X 0,Y 681.397,Z 806.443,A -85,B 0,C 180,E1 4909.027,E2 4909.027} C_VEL
LIN {X 0,Y 679.269,Z 884.881,A -85,B 0,C 180,E1 4910.556,E2 4910.556} C_VEL
LIN {X 0,Y 675.033,Z 956.913,A -85,B 0,C 180,E1 4913.243,E2 4913.243} C_VEL
LIN {X 0,Y 669.758,Z 1025.772,A -85,B 0,C 180,E1 4917.224,E2 4917.224} C_VEL
LIN {X 0,Y 664.885,Z 1086.922,A -85,B 0,C 180,E1 4922.33,E2 4922.33} C_VEL
LIN {X 0,Y 661.427,Z 1136.561,A -85,B 0,C 180,E1 4928.169,E2 4928.169} C_VEL
LIN {X 0,Y 659.69,Z 1171.597,A -85,B 0,C 180,E1 4934.014,E2 4934.014} C_VEL
LIN {X 0,Y 659.014,Z 1194.398,A -85,B 0,C 180,E1 4939.757,E2 4939.757} C_VEL
LIN {X 0,Y 658.863,Z 1206.866,A -85,B 0,C 180,E1 4945.412,E2 4945.412} C_VEL
LIN {X 0,Y 659.032,Z 1209.852,A -85,B 0,C 180,E1 4950.695,E2 4950.695} C_VEL
LIN {X 0,Y 658.951,Z 1203.454,A -85,B 0,C 180,E1 4956.647,E2 4956.647} C_VEL
LIN {X 0,Y 659.253,Z 1186.053,A -85,B 0,C 180,E1 4962.666,E2 4962.666} C_VEL
LIN {X 0,Y 660.281,Z 1158.289,A -85,B 0,C 180,E1 4968.457,E2 4968.457} C_VEL
LIN {X 0,Y 662.967,Z 1115.486,A -85,B 0,C 180,E1 4974.547,E2 4974.547} C_VEL
LIN {X 0,Y 667.268,Z 1058.232,A -85,B 0,C 180,E1 4980.284,E2 4980.284} C_VEL
LIN {X 0,Y 672.538,Z 991.135,A -85,B 0,C 180,E1 4984.974,E2 4984.974} C_VEL
LIN {X 0,Y 677.424,Z 919.959,A -85,B 0,C 180,E1 4988.302,E2 4988.302} C_VEL
LIN {X 0,Y 680.742,Z 845.599,A -85,B 0,C 180,E1 4990.368,E2 4990.368} C_VEL
LIN {X 0,Y 680.062,Z 802.483,A -85,B 0,C 180,E1 4991.125,E2 4991.125} C_VEL
LIN {X 0,Y 658.471,Z 762.06,A -85,B 0,C 180,E1 4993.406,E2 4993.406} C_VEL
LIN {X 0,Y 658.581,Z 762.06,A -85,B 0,C 180,E1 5002.7,E2 5002.7} C_VEL
LIN {X 0,Y 658.752,Z 762.06,A -85,B 0,C 180,E1 5010.273,E2 5010.273} C_VEL
LIN {X 0,Y 658.394,Z 762.06,A -85,B 0,C 180,E1 5017.61,E2 5017.61} C_VEL
LIN {X 0,Y 658.43,Z 762.06,A -85,B 0,C 180,E1 5025.958,E2 5025.958} C_VEL
LIN {X 0,Y 658.844,Z 762.06,A -85,B 0,C 180,E1 5032.684,E2 5032.684} C_VEL
LIN {X 0,Y 658.827,Z 762.06,A -85,B 0,C 180,E1 5040.621,E2 5040.621} C_VEL
LIN {X 0,Y 658.582,Z 762.06,A -85,B 0,C 180,E1 5048.573,E2 5048.573} C_VEL
LIN {X 0,Y 658.3,Z 762.06,A -85,B 0,C 180,E1 5056.704,E2 5056.704} C_VEL
LIN {X 0,Y 658.46,Z 762.06,A -85,B 0,C 180,E1 5064.379,E2 5064.379} C_VEL
LIN {X 0,Y 658.264,Z 762.06,A -85,B 0,C 180,E1 5072.751,E2 5072.751} C_VEL
LIN {X 0,Y 658.134,Z 762.06,A -85,B 0,C 180,E1 5081.023,E2 5081.023} C_VEL
LIN {X 0,Y 658.512,Z 763.799,A -85,B 0,C 180,E1 5087.045,E2 5087.045} C_VEL
LIN {X 0,Y 681.175,Z 806.776,A -85,B 0,C 180,E1 5089.436,E2 5089.436} C_VEL
LIN {X 0,Y 677.947,Z 878.842,A -85,B 0,C 180,E1 5091.257,E2 5091.257} C_VEL
LIN {X 0,Y 673.186,Z 951.708,A -85,B 0,C 180,E1 5094.453,E2 5094.453} C_VEL
LIN {X 0,Y 667.87,Z 1019.634,A -85,B 0,C 180,E1 5098.964,E2 5098.964} C_VEL
LIN {X 0,Y 663.418,Z 1077.964,A -85,B 0,C 180,E1 5104.516,E2 5104.516} C_VEL
LIN {X 0,Y 660.664,Z 1122.386,A -85,B 0,C 180,E1 5110.511,E2 5110.511} C_VEL
LIN {X 0,Y 659.424,Z 1152.158,A -85,B 0,C 180,E1 5116.322,E2 5116.322} C_VEL
LIN {X 0,Y 659.254,Z 1170.659,A -85,B 0,C 180,E1 5122.027,E2 5122.027} C_VEL
LIN {X 0,Y 658.963,Z 1179.385,A -85,B 0,C 180,E1 5127.986,E2 5127.986} C_VEL
LIN {X 0,Y 659.328,Z 1178.37,A -85,B 0,C 180,E1 5133.263,E2 5133.263} C_VEL
LIN {X 0,Y 659.073,Z 1165.297,A -85,B 0,C 180,E1 5139.907,E2 5139.907} C_VEL
LIN {X 0,Y 659.789,Z 1141.332,A -85,B 0,C 180,E1 5145.983,E2 5145.983} C_VEL
LIN {X 0,Y 661.842,Z 1102.386,A -85,B 0,C 180,E1 5152.367,E2 5152.367} C_VEL
LIN {X 0,Y 665.505,Z 1050.053,A -85,B 0,C 180,E1 5158.293,E2 5158.293} C_VEL
LIN {X 0,Y 670.617,Z 985.242,A -85,B 0,C 180,E1 5163.443,E2 5163.443} C_VEL
LIN {X 0,Y 675.758,Z 915.847,A -85,B 0,C 180,E1 5167.212,E2 5167.212} C_VEL
LIN {X 0,Y 679.865,Z 841.574,A -85,B 0,C 180,E1 5169.746,E2 5169.746} C_VEL
LIN {X 0,Y 679.971,Z 801.619,A -85,B 0,C 180,E1 5170.65,E2 5170.65} C_VEL
LIN {X 0,Y 658.587,Z 762.06,A -85,B 0,C 180,E1 5173.013,E2 5173.013} C_VEL
LIN {X 0,Y 658.66,Z 762.06,A -85,B 0,C 180,E1 5182.575,E2 5182.575} C_VEL
LIN {X 0,Y 659.182,Z 763.234,A -85,B 0,C 180,E1 5185.328,E2 5185.328} C_VEL
LIN {X 0,Y 662.238,Z 799.694,A -85,B 0,C 180,E1 5186.866,E2 5186.866} C_VEL
LIN {X 0,Y 661.25,Z 847.602,A -85,B 0,C 180,E1 5188.616,E2 5188.616} C_VEL
LIN {X 0,Y 661.628,Z 974.725,A -85,B 0,C 180,E1 5190.229,E2 5190.229} C_VEL
LIN {X 0,Y 660.934,Z 1013.905,A -85,B 0,C 180,E1 5192.037,E2 5192.037} C_VEL
LIN {X 0,Y 660.154,Z 1043.684,A -85,B 0,C 180,E1 5194.88,E2 5194.88} C_VEL
LIN {X 0,Y 659.783,Z 1060.167,A -85,B 0,C 180,E1 5198.191,E2 5198.191} C_VEL
LIN {X 0,Y 659.804,Z 1063.756,A -85,B 0,C 180,E1 5201.955,E2 5201.955} C_VEL
LIN {X 0,Y 660.31,Z 1052.198,A -85,B 0,C 180,E1 5205.739,E2 5205.739} C_VEL
LIN {X 0,Y 660.55,Z 1026.58,A -85,B 0,C 180,E1 5208.948,E2 5208.948} C_VEL
LIN {X 0,Y 661.38,Z 990.618,A -85,B 0,C 180,E1 5211.144,E2 5211.144} C_VEL
LIN {X 0,Y 661.637,Z 948.363,A -85,B 0,C 180,E1 5212.172,E2 5212.172} C_VEL
LIN {X 0,Y 661.632,Z 838.49,A -85,B 0,C 180,E1 5213.536,E2 5213.536} C_VEL
LIN {X 0,Y 660.139,Z 764.183,A -85,B 0,C 180,E1 5216.512,E2 5216.512} C_VEL
LIN {X 0,Y 659.204,Z 762.06,A -85,B 0,C 180,E1 5218.06,E2 5218.06} C_VEL
LIN {X 0,Y 658.902,Z 762.06,A -85,B 0,C 180,E1 5225.987,E2 5225.987} C_VEL
LIN {X 0,Y 658.618,Z 762.06,A -85,B 0,C 180,E1 5234.038,E2 5234.038} C_VEL
LIN {X 0,Y 658.291,Z 762.06,A -85,B 0,C 180,E1 5242.394,E2 5242.394} C_VEL
LIN {X 0,Y 658.343,Z 762.06,A -85,B 0,C 180,E1 5250.268,E2 5250.268} C_VEL
LIN {X 0,Y 658.066,Z 762.06,A -85,B 0,C 180,E1 5252.818,E2 5252.818} C_VEL
LIN {X 0,Y 650.261,Z 762.06,A -85,B 0,C 180,E1 5255.859,E2 5255.859} C_VEL
LIN {X 0,Y 650.375,Z 762.06,A -85,B 0,C 180,E1 5265.933,E2 5265.933} C_VEL
LIN {X 0,Y 675.28,Z 810.95,A -85,B 0,C 180,E1 5268.638,E2 5268.638} C_VEL
LIN {X 0,Y 672.77,Z 889.719,A -85,B 0,C 180,E1 5270.26,E2 5270.26} C_VEL
LIN {X 0,Y 668.127,Z 961.451,A -85,B 0,C 180,E1 5273.043,E2 5273.043} C_VEL
LIN {X 0,Y 662.354,Z 1030.639,A -85,B 0,C 180,E1 5277.184,E2 5277.184} C_VEL
LIN {X 0,Y 657.012,Z 1092.531,A -85,B 0,C 180,E1 5282.565,E2 5282.565} C_VEL
LIN {X 0,Y 653.404,Z 1140.292,A -85,B 0,C 180,E1 5288.433,E2 5288.433} C_VEL
LIN {X 0,Y 651.688,Z 1173.224,A -85,B 0,C 180,E1 5294.16,E2 5294.16} C_VEL
LIN {X 0,Y 650.969,Z 1195.416,A -85,B 0,C 180,E1 5299.968,E2 5299.968} C_VEL
LIN {X 0,Y 650.881,Z 1206.865,A -85,B 0,C 180,E1 5305.355,E2 5305.355} C_VEL
LIN {X 0,Y 651.026,Z 1209.854,A -85,B 0,C 180,E1 5310.703,E2 5310.703} C_VEL
LIN {X 0,Y 650.963,Z 1203.454,A -85,B 0,C 180,E1 5316.728,E2 5316.728} C_VEL
LIN {X 0,Y 651.33,Z 1187.527,A -85,B 0,C 180,E1 5322.436,E2 5322.436} C_VEL
LIN {X 0,Y 652.382,Z 1158.505,A -85,B 0,C 180,E1 5328.65,E2 5328.65} C_VEL
LIN {X 0,Y 655.301,Z 1115.487,A -85,B 0,C 180,E1 5334.853,E2 5334.853} C_VEL
LIN {X 0,Y 660.028,Z 1058.05,A -85,B 0,C 180,E1 5340.669,E2 5340.669} C_VEL
LIN {X 0,Y 665.728,Z 991.308,A -85,B 0,C 180,E1 5345.374,E2 5345.374} C_VEL
LIN {X 0,Y 670.992,Z 920.681,A -85,B 0,C 180,E1 5348.707,E2 5348.707} C_VEL
LIN {X 0,Y 674.642,Z 845.383,A -85,B 0,C 180,E1 5350.814,E2 5350.814} C_VEL
LIN {X 0,Y 674.08,Z 805.819,A -85,B 0,C 180,E1 5351.524,E2 5351.524} C_VEL
LIN {X 0,Y 651.014,Z 765.079,A -85,B 0,C 180,E1 5354.04,E2 5354.04} C_VEL
LIN {X 0,Y 650.443,Z 762.06,A -85,B 0,C 180,E1 5355.407,E2 5355.407} C_VEL
LIN {X 0,Y 650.574,Z 762.06,A -85,B 0,C 180,E1 5363.636,E2 5363.636} C_VEL
LIN {X 0,Y 650.667,Z 762.06,A -85,B 0,C 180,E1 5371.399,E2 5371.399} C_VEL
LIN {X 0,Y 650.164,Z 762.06,A -85,B 0,C 180,E1 5378.752,E2 5378.752} C_VEL
LIN {X 0,Y 650.446,Z 762.06,A -85,B 0,C 180,E1 5385.782,E2 5385.782} C_VEL
LIN {X 0,Y 650.877,Z 762.06,A -85,B 0,C 180,E1 5392.594,E2 5392.594} C_VEL
LIN {X 0,Y 650.82,Z 762.06,A -85,B 0,C 180,E1 5400.629,E2 5400.629} C_VEL
LIN {X 0,Y 650.551,Z 762.06,A -85,B 0,C 180,E1 5408.68,E2 5408.68} C_VEL
LIN {X 0,Y 650.253,Z 762.06,A -85,B 0,C 180,E1 5416.917,E2 5416.917} C_VEL
LIN {X 0,Y 650.53,Z 762.06,A -85,B 0,C 180,E1 5424.046,E2 5424.046} C_VEL
LIN {X 0,Y 650.365,Z 762.06,A -85,B 0,C 180,E1 5431.616,E2 5431.616} C_VEL
LIN {X 0,Y 650.181,Z 762.06,A -85,B 0,C 180,E1 5439.87,E2 5439.87} C_VEL
LIN {X 0,Y 650.606,Z 763.906,A -85,B 0,C 180,E1 5446.396,E2 5446.396} C_VEL
LIN {X 0,Y 674.994,Z 810.125,A -85,B 0,C 180,E1 5449.055,E2 5449.055} C_VEL
LIN {X 0,Y 671.442,Z 882.33,A -85,B 0,C 180,E1 5450.945,E2 5450.945} C_VEL
LIN {X 0,Y 666.328,Z 953.326,A -85,B 0,C 180,E1 5454.13,E2 5454.13} C_VEL
LIN {X 0,Y 660.553,Z 1021.367,A -85,B 0,C 180,E1 5458.732,E2 5458.732} C_VEL
LIN {X 0,Y 655.708,Z 1079.674,A -85,B 0,C 180,E1 5464.404,E2 5464.404} C_VEL
LIN {X 0,Y 652.642,Z 1124.537,A -85,B 0,C 180,E1 5470.615,E2 5470.615} C_VEL
LIN {X 0,Y 651.356,Z 1153.513,A -85,B 0,C 180,E1 5476.493,E2 5476.493} C_VEL
LIN {X 0,Y 650.971,Z 1172.145,A -85,B 0,C 180,E1 5482.599,E2 5482.599} C_VEL
LIN {X 0,Y 650.968,Z 1179.382,A -85,B 0,C 180,E1 5487.961,E2 5487.961} C_VEL
LIN {X 0,Y 651.303,Z 1178.368,A -85,B 0,C 180,E1 5493.303,E2 5493.303} C_VEL
LIN {X 0,Y 651.303,Z 1167.179,A -85,B 0,C 180,E1 5499.35,E2 5499.35} C_VEL
LIN {X 0,Y 651.892,Z 1143.023,A -85,B 0,C 180,E1 5505.835,E2 5505.835} C_VEL
LIN {X 0,Y 653.991,Z 1104.717,A -85,B 0,C 180,E1 5512.311,E2 5512.311} C_VEL
LIN {X 0,Y 657.934,Z 1052.734,A -85,B 0,C 180,E1 5518.373,E2 5518.373} C_VEL
LIN {X 0,Y 663.345,Z 989.486,A -85,B 0,C 180,E1 5523.551,E2 5523.551} C_VEL
LIN {X 0,Y 668.946,Z 919.536,A -85,B 0,C 180,E1 5527.474,E2 5527.474} C_VEL
LIN {X 0,Y 673.478,Z 845.716,A -85,B 0,C 180,E1 5530.085,E2 5530.085} C_VEL
LIN {X 0,Y 673.614,Z 804.279,A -85,B 0,C 180,E1 5531.071,E2 5531.071} C_VEL
LIN {X 0,Y 650.441,Z 762.06,A -85,B 0,C 180,E1 5533.697,E2 5533.697} C_VEL
LIN {X 0,Y 650.605,Z 762.06,A -85,B 0,C 180,E1 5541.88,E2 5541.88} C_VEL
LIN {X 0,Y 651.229,Z 763.836,A -85,B 0,C 180,E1 5545.155,E2 5545.155} C_VEL
LIN {X 0,Y 654.513,Z 799.437,A -85,B 0,C 180,E1 5546.675,E2 5546.675} C_VEL
LIN {X 0,Y 653.44,Z 850.193,A -85,B 0,C 180,E1 5548.498,E2 5548.498} C_VEL
LIN {X 0,Y 653.775,Z 975.651,A -85,B 0,C 180,E1 5550.114,E2 5550.114} C_VEL
LIN {X 0,Y 653.073,Z 1014.631,A -85,B 0,C 180,E1 5551.924,E2 5551.924} C_VEL
LIN {X 0,Y 652.25,Z 1044.031,A -85,B 0,C 180,E1 5554.719,E2 5554.719} C_VEL
LIN {X 0,Y 651.872,Z 1061.54,A -85,B 0,C 180,E1 5558.275,E2 5558.275} C_VEL
LIN {X 0,Y 651.864,Z 1065.016,A -85,B 0,C 180,E1 5561.727,E2 5561.727} C_VEL
LIN {X 0,Y 652.304,Z 1055.361,A -85,B 0,C 180,E1 5565.362,E2 5565.362} C_VEL
LIN {X 0,Y 652.686,Z 1031.79,A -85,B 0,C 180,E1 5568.644,E2 5568.644} C_VEL
LIN {X 0,Y 653.487,Z 997.599,A -85,B 0,C 180,E1 5570.993,E2 5570.993} C_VEL
LIN {X 0,Y 653.833,Z 956.527,A -85,B 0,C 180,E1 5572.204,E2 5572.204} C_VEL
LIN {X 0,Y 653.874,Z 838.675,A -85,B 0,C 180,E1 5573.711,E2 5573.711} C_VEL
LIN {X 0,Y 652.428,Z 765.727,A -85,B 0,C 180,E1 5576.646,E2 5576.646} C_VEL
LIN {X 0,Y 651.704,Z 762.06,A -85,B 0,C 180,E1 5577.036,E2 5577.036} C_VEL
LIN {X 0,Y 650.858,Z 762.06,A -85,B 0,C 180,E1 5586.061,E2 5586.061} C_VEL
LIN {X 0,Y 650.404,Z 762.06,A -85,B 0,C 180,E1 5594.639,E2 5594.639} C_VEL
LIN {X 0,Y 650.172,Z 762.06,A -85,B 0,C 180,E1 5602.896,E2 5602.896} C_VEL
LIN {X 0,Y 650.388,Z 762.06,A -85,B 0,C 180,E1 5610.149,E2 5610.149} C_VEL
LIN {X 0,Y 650.261,Z 762.06,A -85,B 0,C 180,E1 5615.859,E2 5615.859} C_VEL
